      CALL FC    48 (
           UnitNo                   := #UnitNo,
           PrId                     := #Prid,
           Run                      := DB1941.DBX   17.4,
           PrIdTransfer             := TRUE,
           Start                    := TRUE,
           RetVal                   := #wRetVal);
Strt: NOP   0;

      L     0;
      T     DB502.DBD  156;

NETWORK
TITLE =external releases

      SET   ;
      =     DB2940.DBX  106.7;
      =     DB2940.DBX  266.7;
      =     DB2940.DBX  346.7;
      =     DB2940.DBX  426.7;
      =     DB2940.DBX  506.7;
      =     DB2940.DBX  586.7;
      =     DB2940.DBX  666.7;
      =     DB2940.DBX  746.7;
      =     DB2940.DBX  826.7;
      =     DB2940.DBX  906.7;
      =     DB2940.DBX  986.7;
      =     DB2940.DBX 1066.7;
      =     DB2940.DBX 1146.7;
      =     DB2940.DBX 1226.7;
      =     DB2940.DBX 1306.7;
      =     DB2940.DBX 1386.7;
      =     DB2940.DBX 1466.7;
      =     DB2940.DBX 1546.7;
NETWORK
TITLE =write own unit data

      SET   ;

//-- CIP Communication ---------------------------------------
      AN    DB1941.DBX   15.0;
      AN    DB1941.DBX 1233.6; // CIP Active (Slave)
      A     #ComCIP;
      JCN   NCIP;
//Conductivity CIP Return
      L     DB1945.DBD  150;
      T     DB1941.DBD  626;

//Temperature CIP Return
      L     DB1945.DBD  146;
      T     DB1941.DBD  594;

//CIP Prerun Pump SP
      CALL FC    45 (
           SFM                      := DB1941.DBD  686,
           Indexes                  := #SFM36);


      L     0.000000e+000;
      A     #SFM36.I01;
      =     DB1945.DBX  171.7;
      JCN   pfc;
      L     DB1941.DBD  654;
pfc:  NOP   0;
      A     #SFM36.I02;
      =     DB1945.DBX  172.0;
      JCN   ppc;
      L     DB1941.DBD  670;
ppc:  NOP   0;
      A     #SFM36.I03;
      =     DB1945.DBX  171.6;
      JCN   pxc;
      L     DB1941.DBD  574;
pxc:  NOP   0;
      T     DB1945.DBD  182;

//CIP Return
      L     DB1941.DBD  558;
      T     DB1945.DBD  186;
      L     DB1945.DBD  138;
      T     DB1941.DBD  562;

//CIP Prerun
      L     DB1941.DBD  542;
      T     DB1945.DBD  190;
      L     DB1945.DBD  142;
      T     DB1941.DBD  546;

// CIP Prerun Temperature
      L     DB1941.DBD  686;
      T     DB1945.DBD  182;

// Write Own Data to CIP
      L     DB1945.DBD   10;
      T     DB1945.DBD  154;

      L     DB1945.DBW   14;
      T     DB1945.DBW  158;

      L     DB1945.DBW   16;
      T     DB1945.DBW  160;

      L     DB1945.DBW   18;
      T     DB1945.DBW  162;

      L     DB1945.DBW   20;
      T     DB1945.DBW  164;

      L     DB1945.DBW   22;
      T     DB1945.DBW  166;

      A     DB1945.DBX   24.0;
      =     DB1945.DBX  168.0;

      A     DB1945.DBX   24.1;
      =     DB1945.DBX  168.1;

      A     DB1945.DBX   24.2;
      =     DB1945.DBX  168.2;

      A     DB1945.DBX   24.3;
      =     DB1945.DBX  168.3;

      A     DB1945.DBX   24.4;
      =     DB1945.DBX  168.4;

      A     DB1945.DBX   24.5;
      =     DB1945.DBX  168.5;

      A     DB1945.DBX   24.6;
      =     DB1945.DBX  168.6;

      A     DB1945.DBX   24.7;
      =     DB1945.DBX  168.7;

      L     DB1945.DBD  138; // CIP Amount
      T     DB1945.DBD   54; // CIP Amount

// Copy Data to CIP
      CALL SFC   20 (
           SRCBLK                   := DB1945.ToCIP,
           RET_VAL                  := #iRetVal,
           DSTBLK                   := DB502.ToCIP1);

      CLR   ;
      =     DB1945.DBX  173.7;

NCIP: NOP   0;

//Empty Signal
//A     "U094SpID".SpI.Sig //!!!! Insert correct Empty Signal !!!
      CLR   ;
      =     DB1945.DBX   26.5;

//Full Signal
//A     "U094SpID".SpI.Sig //!!!! Insert correct Full Signal !!!
      CLR   ;
      =     DB1945.DBX   26.2;

//CIP Program Selected
      A     #CIP;
      =     DB1945.DBX   27.1;

// Emergency Stop
      A     #EStopOK; //If needed add or replace with own SpI
      =     DB1945.DBX   27.0; //Emergency Stop OK


NETWORK
TITLE = read from other unit data



END_FUNCTION_BLOCK

FUNCTION_BLOCK FB 1949
TITLE =U094: CIP 1 Distribution
AUTHOR : Woermann
FAMILY : BOTEC_F1
NAME : Sim
VERSION : 0.1


VAR_TEMP
  CIP : BOOL ;	//CIP active
  xTmp : BOOL ;	//Temporary BOOL (free for general use)
  iTmp : INT ;	//Temporary INT (free for general use)
  rTmp : REAL ;	//Temporary REAL (free for general use)
  UnitNo : INT ;	//Unit Number
END_VAR
BEGIN
NETWORK
TITLE =General

      SET   ;
// get unit number ----------------------------------------------------------
      L     DB1940.DBW    0;
      T     #UnitNo;

// CIP ----------------------------------------------------------------------
      L     DB1941.DBD   54;
      L     0;
      <D    ;
      =     #CIP;

NETWORK
TITLE =Actuator

      A     DB1941.DBX   17.3;
      =     DB2940.DBX  105.3;
      =     DB2940.DBX  265.3;
      =     DB2940.DBX  345.3;
      =     DB2940.DBX  425.3;
      =     DB2940.DBX  505.3;
      =     DB2940.DBX  585.3;
      =     DB2940.DBX  665.3;
      =     DB2940.DBX  745.3;
      =     DB2940.DBX  825.3;
      =     DB2940.DBX  905.3;
      =     DB2940.DBX  985.3;
      =     DB2940.DBX 1065.3;
      =     DB2940.DBX 1145.3;
      =     DB2940.DBX 1225.3;
      =     DB2940.DBX 1305.3;
      =     DB2940.DBX 1385.3;
      =     DB2940.DBX 1465.3;
      =     DB2940.DBX 1545.3;


NETWORK
TITLE =Special Input

      A     DB1941.DBX   17.3;
      =     DB2941.DBX   81.3;
      =     DB2941.DBX  141.3;
      =     DB2941.DBX  201.3;
      =     DB2941.DBX  261.3;
      =     DB2941.DBX  321.3;
      =     DB2941.DBX  381.3;

NETWORK
TITLE =Counter

      A     DB1941.DBX   17.3;
      A     M    101.0;


      CLR   ;
NETWORK
TITLE =Analog Input

      A     DB1941.DBX   17.3;

NETWORK
TITLE =Universal Value

      A     DB1941.DBX   17.3;
//      =     "U094UnVD".unv001.Sim;
//      =     "U094UnVD".unv002.Sim;
//      =     "U094UnVD".RK1_KreisNr.Sim
//      =     "U094UnVD".RK1_Medium.Sim

NETWORK
TITLE =PID

      A     DB1941.DBX   17.3;

NETWORK
TITLE =Message

      A     DB1941.DBX   17.3;
//      =     "U094MsgD".msg001.Sim;
//      =     "U094MsgD".msg002.Sim;

NETWORK
TITLE =VLT

      A     DB1941.DBX   17.3;

END_FUNCTION_BLOCK

FUNCTION_BLOCK FB 1955
TITLE =U095: CIP 2 Distribution
FAMILY : BOTEC_F1
NAME : Comm
VERSION : 0.1


VAR_TEMP
  iRetVal : INT ;	//return value as integer
  wRetVal : WORD ;	//return value as word
  Run : BOOL ;	//Unit in "RUN" mode
  EStopOK : BOOL ;	//Emergency Stop OK
  CIP : BOOL ;	//CIP Program Selected
  ComCIP : BOOL ;	//Communication with CIP Active
  xTmp : BOOL ;	//Temporary BOOL (free for general use)
  iTmp : INT ;	//Temporary INT (free for general use)
  rTmp : REAL ;	//Temporary REAL (free for general use)
  dTmp : DINT ;	//Temporary DINT (free for general use)
  UnitNo : INT ;	//Unit Number
  EquipmentID : INT ;	//Equipment ID
  Prid : DINT ;	//Process ID
  SFM36 : STRUCT 	// CIP Pump Mode
   I00 : BOOL ;	// Off
   I01 : BOOL ;	// Flow
   I02 : BOOL ;	// Pressure
   I03 : BOOL ;	// Fix Speed
   I04 : BOOL ;
   I05 : BOOL ;
   I06 : BOOL ;
   I07 : BOOL ;
   I08 : BOOL ;
   I09 : BOOL ;
   I10 : BOOL ;
   I11 : BOOL ;
   I12 : BOOL ;
   I13 : BOOL ;
   I14 : BOOL ;
   I15 : BOOL ;
   I16 : BOOL ;
   I17 : BOOL ;
   I18 : BOOL ;
   I19 : BOOL ;
   I20 : BOOL ;
   I21 : BOOL ;
   I22 : BOOL ;
   I23 : BOOL ;
   I24 : BOOL ;
   I25 : BOOL ;
   I26 : BOOL ;
   I27 : BOOL ;
   I28 : BOOL ;
   I29 : BOOL ;
   I30 : BOOL ;
   I31 : BOOL ;
  END_STRUCT ;
END_VAR
BEGIN
NETWORK
TITLE =general

      SET   ;

// unit & equipment number ---------------------------------------------------
      L     DB1950.DBW    0;
      T     #UnitNo;

      L     DB1955.DBW   14;
      L     1000;
      *I    ;
      L     #UnitNo;
      +I    ;
      T     #EquipmentID;

// CIP ----------------------------------------------------------------------
      L     DB1955.DBW   18;
      L     0;
      <I    ;
      =     #CIP;

// Communicating Units-------------------------------------------------------
      L     DB1955.DBD   10;
      L     DB1955.DBD  106;
      ==D   ;
      =     #ComCIP;

// emergency OK -------------------------------------------------------------
      A     DB1955.DBX   75.0; //General Emergency Stop OK
      =     #EStopOK;

NETWORK
TITLE =read other unit's data

      SET   ;

// ... General Unit ----------/

      CALL FC   563 (
           ActReq                   := M    101.0,
           PLCNo                    := DB1955.DBW   14,
           SourceUnitNo             := 99,
           IsTUnit                  := FALSE,
           DstComDRec               := DB1955.GEN,
           RET_VAL                  := #wRetVal);


// ... CIP Unit ------------- /

      CALL FC   563 (
           ActReq                   := M    101.0,
           PLCNo                    := 3,
           SourceUnitNo             := 92,
           IsTUnit                  := FALSE,
           DstComDRec               := DB1955.CIP,
           RET_VAL                  := #wRetVal);

// ... To CIP Unit ------------- /
      AN    DB1951.DBX   15.0;
      A     DB1951.DBX 1233.6; // CIP Active (Slave)
      O     DB1951.DBX 1230.3; // production active
//    A     #ComCIP
      JCN   Slav;
      CALL SFC   20 (
           SRCBLK                   := DB502.ToCIP2,
           RET_VAL                  := #iRetVal,
           DSTBLK                   := DB1955.ToCIP);
Slav: NOP   0;

NETWORK
TITLE =remote start

      SET   ;

//-----------------------------------
// Start Request
//-----------------------------------
      L     DB502.DBD  160;
      L     0;
      >D    ;
      A     DB1951.DBX   15.0;
      A     DB1951.DBX   17.4;
      JCN   Strt;
      L     DB502.DBD  160;
      T     #Prid;

      CALL FC    48 (
           UnitNo                   := #UnitNo,
           PrId                     := #Prid,
           Run                      := DB1951.DBX   17.4,
           PrIdTransfer             := TRUE,
           Start                    := TRUE,
           RetVal                   := #wRetVal);
Strt: NOP   0;

      L     0;
      T     DB502.DBD  160;


NETWORK
TITLE =external releases

      SET   ;
      =     DB2950.DBX  266.7;
      =     DB2950.DBX  346.7;
      =     DB2950.DBX  506.7;
      =     DB2950.DBX  586.7;
NETWORK
TITLE =write own unit data

      SET   ;

//-- CIP Communication ---------------------------------------
      AN    DB1951.DBX   15.0;
      AN    DB1951.DBX 1233.6; // CIP Active (Slave)
      A     #ComCIP;
      JCN   NCIP;
//Conductivity CIP Return
      L     DB1955.DBD  150;
      T     DB1951.DBD  626;

//Temperature CIP Return
      L     DB1955.DBD  146;
      T     DB1951.DBD  594;

//CIP Prerun Pump SP
      CALL FC    45 (
           SFM                      := DB1951.DBD  686,
           Indexes                  := #SFM36);


      L     0.000000e+000;
      A     #SFM36.I01;
      =     DB1955.DBX  171.7;
      JCN   pfc;
      L     DB1951.DBD  654;
pfc:  NOP   0;
      A     #SFM36.I02;
      =     DB1955.DBX  172.0;
      JCN   ppc;
      L     DB1951.DBD  670;
ppc:  NOP   0;
      A     #SFM36.I03;
      =     DB1955.DBX  171.6;
      JCN   pxc;
      L     DB1951.DBD  574;
pxc:  NOP   0;
      T     DB1955.DBD  182;

//CIP Return
      L     DB1951.DBD  558;
      T     DB1955.DBD  186;
      L     DB1955.DBD  138;
      T     DB1951.DBD  562;

//CIP Prerun
      L     DB1951.DBD  542;
      T     DB1955.DBD  190;
      L     DB1955.DBD  142;
      T     DB1951.DBD  546;

// CIP Prerun Temperature
      L     DB1951.DBD  686;
      T     DB1955.DBD  182;

// Write Own Data to CIP
      L     DB1955.DBD   10;
      T     DB1955.DBD  154;

      L     DB1955.DBW   14;
      T     DB1955.DBW  158;

      L     DB1955.DBW   16;
      T     DB1955.DBW  160;

      L     DB1955.DBW   18;
      T     DB1955.DBW  162;

      L     DB1955.DBW   20;
      T     DB1955.DBW  164;

      L     DB1955.DBW   22;
      T     DB1955.DBW  166;

      A     DB1955.DBX   24.0;
      =     DB1955.DBX  168.0;

      A     DB1955.DBX   24.1;
      =     DB1955.DBX  168.1;

      A     DB1955.DBX   24.2;
      =     DB1955.DBX  168.2;

      A     DB1955.DBX   24.3;
      =     DB1955.DBX  168.3;

      A     DB1955.DBX   24.4;
      =     DB1955.DBX  168.4;

      A     DB1955.DBX   24.5;
      =     DB1955.DBX  168.5;

      A     DB1955.DBX   24.6;
      =     DB1955.DBX  168.6;

      A     DB1955.DBX   24.7;
      =     DB1955.DBX  168.7;

      L     DB1955.DBD  138; // CIP Amount
      T     DB1955.DBD   54; // CIP Amount

// Copy Data to CIP
      CALL SFC   20 (
           SRCBLK                   := DB1955.ToCIP,
           RET_VAL                  := #iRetVal,
           DSTBLK                   := DB502.ToCIP2);

NCIP: NOP   0;

//Empty Signal
//A     "U095SpID".SpI.Sig //!!!! Insert correct Empty Signal !!!
      CLR   ;
      =     DB1955.DBX   26.5;

//Full Signal
//A     "U095SpID".SpI.Sig //!!!! Insert correct Full Signal !!!
      CLR   ;
      =     DB1955.DBX   26.2;

//CIP Program Selected
      A     #CIP;
      =     DB1955.DBX   27.1;

// Emergency Stop
      A     #EStopOK; //If needed add or replace with own SpI
      =     DB1955.DBX   27.0; //Emergency Stop OK


NETWORK
TITLE = read from other unit data



END_FUNCTION_BLOCK

FUNCTION_BLOCK FB 1959
TITLE =U095: CIP 2 Distribution
AUTHOR : Woermann
FAMILY : BOTEC_F1
NAME : Sim
VERSION : 0.1


VAR_TEMP
  CIP : BOOL ;	//CIP active
  xTmp : BOOL ;	//Temporary BOOL (free for general use)
  iTmp : INT ;	//Temporary INT (free for general use)
  rTmp : REAL ;	//Temporary REAL (free for general use)
  UnitNo : INT ;	//Unit Number
END_VAR
BEGIN
NETWORK
TITLE =General

      SET   ;
// get unit number ----------------------------------------------------------
      L     DB1950.DBW    0;
      T     #UnitNo;

// CIP ----------------------------------------------------------------------
      L     DB1951.DBD   54;
      L     0;
      <D    ;
      =     #CIP;

NETWORK
TITLE =Actuator

      A     DB1951.DBX   17.3;
      =     DB2950.DBX  265.3;
      =     DB2950.DBX  345.3;
      =     DB2950.DBX  505.3;
      =     DB2950.DBX  585.3;
NETWORK
TITLE =Special Input

      A     DB1951.DBX   17.3;
      =     DB2951.DBX   81.3;
      =     DB2951.DBX  141.3;
      =     DB2951.DBX  201.3;
      =     DB2951.DBX  261.3;
NETWORK
TITLE =Counter

      A     DB1951.DBX   17.3;
      A     M    101.0;


      CLR   ;
NETWORK
TITLE =Analog Input

      A     DB1951.DBX   17.3;

NETWORK
TITLE =Universal Value

      A     DB1951.DBX   17.3;
//      =     "U095UnVD".unv001.Sim;
//      =     "U095UnVD".unv002.Sim;
//      =     "U095UnVD".RK2_KreisNr.Sim;
//      =     "U095UnVD".RK2_Medium.Sim;

NETWORK
TITLE =PID

      A     DB1951.DBX   17.3;

NETWORK
TITLE =Message

      A     DB1951.DBX   17.3;
//      =     "U095MsgD".msg001.Sim;
//      =     "U095MsgD".msg002.Sim;

NETWORK
TITLE =VLT

      A     DB1951.DBX   17.3;

END_FUNCTION_BLOCK

FUNCTION_BLOCK FB 1965
TITLE =U096: CIP 3 Distribution
FAMILY : BOTEC_F1
NAME : Comm
VERSION : 0.1


VAR_TEMP
  iRetVal : INT ;	//return value as integer
  wRetVal : WORD ;	//return value as word
  Run : BOOL ;	//Unit in "RUN" mode
  EStopOK : BOOL ;	//Emergency Stop OK
  CIP : BOOL ;	//CIP Program Selected
  ComCIP : BOOL ;	//Communication with CIP Active
  xTmp : BOOL ;	//Temporary BOOL (free for general use)
  iTmp : INT ;	//Temporary INT (free for general use)
  rTmp : REAL ;	//Temporary REAL (free for general use)
  dTmp : DINT ;	//Temporary DINT (free for general use)
  UnitNo : INT ;	//Unit Number
  EquipmentID : INT ;	//Equipment ID
  Prid : DINT ;	//Process ID
  SFM36 : STRUCT 	// CIP Pump Mode
   I00 : BOOL ;	// Off
   I01 : BOOL ;	// Flow
   I02 : BOOL ;	// Pressure
   I03 : BOOL ;	// Fix Speed
   I04 : BOOL ;
   I05 : BOOL ;
   I06 : BOOL ;
   I07 : BOOL ;
   I08 : BOOL ;
   I09 : BOOL ;
   I10 : BOOL ;
   I11 : BOOL ;
   I12 : BOOL ;
   I13 : BOOL ;
   I14 : BOOL ;
   I15 : BOOL ;
   I16 : BOOL ;
   I17 : BOOL ;
   I18 : BOOL ;
   I19 : BOOL ;
   I20 : BOOL ;
   I21 : BOOL ;
   I22 : BOOL ;
   I23 : BOOL ;
   I24 : BOOL ;
   I25 : BOOL ;
   I26 : BOOL ;
   I27 : BOOL ;
   I28 : BOOL ;
   I29 : BOOL ;
   I30 : BOOL ;
   I31 : BOOL ;
  END_STRUCT ;
END_VAR
BEGIN
NETWORK
TITLE =general

      SET   ;

// unit & equipment number ---------------------------------------------------
      L     DB1960.DBW    0;
      T     #UnitNo;

      L     DB1965.DBW   14;
      L     1000;
      *I    ;
      L     #UnitNo;
      +I    ;
      T     #EquipmentID;

// CIP ----------------------------------------------------------------------
      L     DB1965.DBW   18;
      L     0;
      <I    ;
      =     #CIP;

// Communicating Units-------------------------------------------------------
      L     DB1965.DBD   10;
      L     DB1965.DBD  106;
      ==D   ;
      =     #ComCIP;

// emergency OK -------------------------------------------------------------
      A     DB1965.DBX   75.0; //General Emergency Stop OK
      =     #EStopOK;

NETWORK
TITLE =read other unit's data

      SET   ;

// ... General Unit ----------/

      CALL FC   563 (
           ActReq                   := M    101.0,
           PLCNo                    := DB1965.DBW   14,
           SourceUnitNo             := 99,
           IsTUnit                  := FALSE,
           DstComDRec               := DB1965.GEN,
           RET_VAL                  := #wRetVal);


// ... CIP Unit ------------- /

      CALL FC   563 (
           ActReq                   := M    101.0,
           PLCNo                    := 3,
           SourceUnitNo             := 93,
           IsTUnit                  := FALSE,
           DstComDRec               := DB1965.CIP,
           RET_VAL                  := #wRetVal);

// ... To CIP Unit ------------- /
      A     DB1961.DBX 1233.6; // CIP Active (Slave)
      O     DB1961.DBX 1230.3; // production active
      AN    DB1961.DBX   15.0;

// A     #ComCIP
      JCN   Slav;
      CALL SFC   20 (
           SRCBLK                   := DB502.ToCIP3,
           RET_VAL                  := #iRetVal,
           DSTBLK                   := DB1965.ToCIP);
Slav: NOP   0;
NETWORK
TITLE =remote start

      SET   ;

//-----------------------------------
// Start Request
//-----------------------------------
      L     DB502.DBD  164;
      L     0;
      >D    ;
      A     DB1961.DBX   15.0;
      A     DB1961.DBX   17.4;
      JCN   Strt;
      L     DB502.DBD  164;
      T     #Prid;

      CALL FC    48 (
           UnitNo                   := #UnitNo,
           PrId                     := #Prid,
           Run                      := DB1961.DBX   17.4,
           PrIdTransfer             := TRUE,
           Start                    := TRUE,
           RetVal                   := #wRetVal);
Strt: NOP   0;

      L     0;
      T     DB502.DBD  164;


NETWORK
TITLE =external releases

      SET   ;
      =     DB2960.DBX  186.7;
      =     DB2960.DBX  266.7;
      =     DB2960.DBX  346.7;
      =     DB2960.DBX  426.7;
      =     DB2960.DBX  506.7;
      =     DB2960.DBX  586.7;
      =     DB2960.DBX  666.7;
      =     DB2960.DBX  746.7;
      =     DB2960.DBX  826.7;
      =     DB2960.DBX  906.7;
      =     DB2960.DBX  986.7;
      =     DB2960.DBX 1066.7;
      =     DB2960.DBX 1146.7;
      =     DB2960.DBX 1226.7;
      =     DB2960.DBX 1306.7;
      =     DB2960.DBX 1546.7;
NETWORK
TITLE =write own unit data

      SET   ;

//-- CIP Communication ---------------------------------------
      AN    DB1961.DBX   15.0;
      AN    DB1961.DBX 1233.6; // CIP Active (Slave)
      A     #ComCIP;
      JCN   NCIP;
//Conductivity CIP Return
      L     DB1965.DBD  150;
      T     DB1961.DBD  626;

//Temperature CIP Return
      L     DB1965.DBD  146;
      T     DB1961.DBD  594;

//CIP Prerun Pump SP

      CALL FC    45 (
           SFM                      := DB1961.DBD  686,
           Indexes                  := #SFM36);


      L     0.000000e+000;
      A     #SFM36.I01;
      =     DB1965.DBX  171.7;
      JCN   pfc;
      L     DB1961.DBD  654;
pfc:  NOP   0;
      A     #SFM36.I02;
      =     DB1965.DBX  172.0;
      JCN   ppc;
      L     DB1961.DBD  670;
ppc:  NOP   0;
      A     #SFM36.I03;
      =     DB1965.DBX  171.6;
      JCN   pxc;
      L     DB1961.DBD  574;
pxc:  NOP   0;
      T     DB1965.DBD  182;

//CIP Return
      L     DB1961.DBD  558;
      T     DB1965.DBD  186;
      L     DB1965.DBD  138;
      T     DB1961.DBD  562;

//CIP Prerun
      L     DB1961.DBD  542;
      T     DB1965.DBD  190;
      L     DB1965.DBD  142;
      T     DB1961.DBD  546;

// CIP Prerun Temperature
      L     DB1961.DBD  686;
      T     DB1965.DBD  182;

// Write Own Data to CIP
      L     DB1965.DBD   10;
      T     DB1965.DBD  154;

      L     DB1965.DBW   14;
      T     DB1965.DBW  158;

      L     DB1965.DBW   16;
      T     DB1965.DBW  160;

      L     DB1965.DBW   18;
      T     DB1965.DBW  162;

      L     DB1965.DBW   20;
      T     DB1965.DBW  164;

      L     DB1965.DBW   22;
      T     DB1965.DBW  166;

      A     DB1965.DBX   24.0;
      =     DB1965.DBX  168.0;

      A     DB1965.DBX   24.1;
      =     DB1965.DBX  168.1;

      A     DB1965.DBX   24.2;
      =     DB1965.DBX  168.2;

      A     DB1965.DBX   24.3;
      =     DB1965.DBX  168.3;

      A     DB1965.DBX   24.4;
      =     DB1965.DBX  168.4;

      A     DB1965.DBX   24.5;
      =     DB1965.DBX  168.5;

      A     DB1965.DBX   24.6;
      =     DB1965.DBX  168.6;

      A     DB1965.DBX   24.7;
      =     DB1965.DBX  168.7;

      L     DB1965.DBD  138; // CIP Amount
      T     DB1965.DBD   54; // CIP Amount

// Copy Data to CIP
      CALL SFC   20 (
           SRCBLK                   := DB1965.ToCIP,
           RET_VAL                  := #iRetVal,
           DSTBLK                   := DB502.ToCIP3);

NCIP: NOP   0;

//Empty Signal
//A     "U096SpID".SpI.Sig //!!!! Insert correct Empty Signal !!!
      CLR   ;
      =     DB1965.DBX   26.5;

//Full Signal
//A     "U096SpID".SpI.Sig //!!!! Insert correct Full Signal !!!
      CLR   ;
      =     DB1965.DBX   26.2;

//CIP Program Selected
      A     #CIP;
      =     DB1965.DBX   27.1;

// Emergency Stop
      A     #EStopOK; //If needed add or replace with own SpI
      =     DB1965.DBX   27.0; //Emergency Stop OK


NETWORK
TITLE = read from other unit data



END_FUNCTION_BLOCK

FUNCTION_BLOCK FB 1969
TITLE =U096: CIP 3 Distribution
AUTHOR : Woermann
FAMILY : BOTEC_F1
NAME : Sim
VERSION : 0.1


VAR_TEMP
  CIP : BOOL ;	//CIP active
  xTmp : BOOL ;	//Temporary BOOL (free for general use)
  iTmp : INT ;	//Temporary INT (free for general use)
  rTmp : REAL ;	//Temporary REAL (free for general use)
  UnitNo : INT ;	//Unit Number
END_VAR
BEGIN
NETWORK
TITLE =General

      SET   ;
// get unit number ----------------------------------------------------------
      L     DB1960.DBW    0;
      T     #UnitNo;

// CIP ----------------------------------------------------------------------
      L     DB1961.DBD   54;
      L     0;
      <D    ;
      =     #CIP;

NETWORK
TITLE =Actuator

      A     DB1961.DBX   17.3;
      =     DB2960.DBX  185.3;
      =     DB2960.DBX  265.3;
      =     DB2960.DBX  345.3;
      =     DB2960.DBX  425.3;
      =     DB2960.DBX  505.3;
      =     DB2960.DBX  585.3;
      =     DB2960.DBX  665.3;
      =     DB2960.DBX  745.3;
      =     DB2960.DBX  825.3;
      =     DB2960.DBX  905.3;
      =     DB2960.DBX  985.3;
      =     DB2960.DBX 1065.3;
      =     DB2960.DBX 1145.3;
      =     DB2960.DBX 1225.3;
      =     DB2960.DBX 1305.3;
      =     DB2960.DBX 1545.3;
NETWORK
TITLE =Special Input

      A     DB1961.DBX   17.3;
      =     DB2961.DBX   81.3;
      =     DB2961.DBX  141.3;
      =     DB2961.DBX  201.3;
      =     DB2961.DBX  261.3;
      =     DB2961.DBX  321.3;
      =     DB2961.DBX  381.3;

NETWORK
TITLE =Counter

      A     DB1961.DBX   17.3;
      A     M    101.0;
      CLR   ;
NETWORK
TITLE =Analog Input

      A     DB1961.DBX   17.3;

NETWORK
TITLE =Universal Value

      A     DB1961.DBX   17.3;
//      =     "U096UnVD".unv001.Sim;
//      =     "U096UnVD".unv002.Sim;
//      =     "U096UnVD".RK3_KreisNr.Sim;
//      =     "U096UnVD".RK3_Medium.Sim;

NETWORK
TITLE =PID

      A     DB1961.DBX   17.3;

NETWORK
TITLE =Message

      A     DB1961.DBX   17.3;
//      =     "U096MsgD".msg001.Sim;
//      =     "U096MsgD".msg002.Sim;

NETWORK
TITLE =VLT

      A     DB1961.DBX   17.3;

END_FUNCTION_BLOCK

FUNCTION_BLOCK FB 1985
TITLE =U098: General Syrup Room
FAMILY : BOTEC_F1
NAME : Comm
VERSION : 0.1


VAR_TEMP
  iRetVal : INT ;	//return value as integer
  wRetVal : WORD ;	//return value as word
  Run : BOOL ;	//Unit in "RUN" mode
  EStopOK : BOOL ;	//Emergency Stop OK
  CIP : BOOL ;	//CIP Program Selected
  ComCIP : BOOL ;	//Communication with CIP Active
  xTmp : BOOL ;	//Temporary BOOL (free for general use)
  iTmp : INT ;	//Temporary INT (free for general use)
  rTmp : REAL ;	//Temporary REAL (free for general use)
  dTmp : DINT ;	//Temporary DINT (free for general use)
  UnitNo : INT ;	//Unit Number
  EquipmentID : INT ;	//Equipment ID
  Prid : DINT ;	//Process ID
  SFM36 : STRUCT 	// CIP Pump Mode
   I00 : BOOL ;	// Off
   I01 : BOOL ;	// Flow
   I02 : BOOL ;	// Pressure
   I03 : BOOL ;	// Fix Speed
   I04 : BOOL ;
   I05 : BOOL ;
   I06 : BOOL ;
   I07 : BOOL ;
   I08 : BOOL ;
   I09 : BOOL ;
   I10 : BOOL ;
   I11 : BOOL ;
   I12 : BOOL ;
   I13 : BOOL ;
   I14 : BOOL ;
   I15 : BOOL ;
   I16 : BOOL ;
   I17 : BOOL ;
   I18 : BOOL ;
   I19 : BOOL ;
   I20 : BOOL ;
   I21 : BOOL ;
   I22 : BOOL ;
   I23 : BOOL ;
   I24 : BOOL ;
   I25 : BOOL ;
   I26 : BOOL ;
   I27 : BOOL ;
   I28 : BOOL ;
   I29 : BOOL ;
   I30 : BOOL ;
   I31 : BOOL ;
  END_STRUCT ;
END_VAR
BEGIN
NETWORK
TITLE =general

      SET   ;

// unit & equipment number ---------------------------------------------------
      L     DB1980.DBW    0;
      T     #UnitNo;

      L     DB1985.DBW   14;
      L     1000;
      *I    ;
      L     #UnitNo;
      +I    ;
      T     #EquipmentID;

// CIP ----------------------------------------------------------------------
      L     DB1985.DBW   18;
      L     0;
      <I    ;
      =     #CIP;

// Communicating Units-------------------------------------------------------
      L     DB1985.DBD   10;
      L     DB1985.DBD  106;
      ==D   ;
      =     #ComCIP;

// emergency OK -------------------------------------------------------------
      A     DB1985.DBX   75.0; //General Emergency Stop OK
      =     #EStopOK;

NETWORK
TITLE =read other unit's data

      SET   ;

// ... General Unit ----------/

      CALL FC   563 (
           ActReq                   := M    101.0,
           PLCNo                    := DB1985.DBW   14,
           SourceUnitNo             := 99,
           IsTUnit                  := FALSE,
           DstComDRec               := DB1985.GEN,
           RET_VAL                  := #wRetVal);


NETWORK
TITLE =remote start

      SET   ;
// !!! insert correct condition of unit start !!!
      A     DB1981.DBX   15.0;
      A     DB1981.DBX   17.4;
      CLR   ;
      JCN   Strt;
      L     DB1985.DBD   10;
//L        L#-1;                            // Prid negative to start on its own
      T     #Prid;

      CALL FC    48 (
           UnitNo                   := #UnitNo,
           PrId                     := #Prid,
           Run                      := DB1981.DBX   17.4,
           PrIdTransfer             := TRUE,
           Start                    := TRUE,
           RetVal                   := #wRetVal);
Strt: NOP   0;
NETWORK
TITLE =external releases

      SET   ;
      =     DB2980.DBX  106.7;
      =     DB2980.DBX  186.7;
      =     DB2980.DBX  266.7;
      =     DB2980.DBX  346.7;
      =     DB2980.DBX  426.7;
      =     DB2980.DBX  506.7;
      =     DB2980.DBX  586.7;
      =     DB2980.DBX  666.7;
NETWORK
TITLE =write own unit data

      SET   ;

//-- CIP Communication ---------------------------------------
      AN    DB1981.DBX   15.0;
//      AN "U098SeqD".Seq.PO.B30 // CIP Active (Slave)
      A     #ComCIP;
      JCN   NCIP;
//Conductivity CIP Return
      L     DB1985.DBD  150;
      T     DB1981.DBD  626;

//Temperature CIP Return
      L     DB1985.DBD  146;
      T     DB1981.DBD  594;

//CIP Prerun Pump SP

      CALL FC    45 (
           SFM                      := DB1981.DBD  686,
           Indexes                  := #SFM36);


      L     0.000000e+000;
      A     #SFM36.I01;
      =     DB1985.DBX  171.7;
      JCN   pfc;
      L     DB1981.DBD  654;
pfc:  NOP   0;
      A     #SFM36.I02;
      =     DB1985.DBX  172.0;
      JCN   ppc;
      L     DB1981.DBD  670;
ppc:  NOP   0;
      A     #SFM36.I03;
      =     DB1985.DBX  171.6;
      JCN   pxc;
      L     DB1981.DBD  574;
pxc:  NOP   0;
      T     DB1985.DBD  182;

//CIP Return
      L     DB1981.DBD  558;
      T     DB1985.DBD  186;
      L     DB1985.DBD  138;
      T     DB1981.DBD  562;

//CIP Prerun
      L     DB1981.DBD  542;
      T     DB1985.DBD  190;
      L     DB1985.DBD  142;
      T     DB1981.DBD  546;

// Write Own Data to CIP
      L     DB1985.DBD   10;
      T     DB1985.DBD  154;

      L     DB1985.DBW   14;
      T     DB1985.DBW  158;

      L     DB1985.DBW   16;
      T     DB1985.DBW  160;

      L     DB1985.DBW   18;
      T     DB1985.DBW  162;

      L     DB1985.DBW   20;
      T     DB1985.DBW  164;

      L     DB1985.DBW   22;
      T     DB1985.DBW  166;

      A     DB1985.DBX   24.0;
      =     DB1985.DBX  168.0;

      A     DB1985.DBX   24.1;
      =     DB1985.DBX  168.1;

      A     DB1985.DBX   24.2;
      =     DB1985.DBX  168.2;

      A     DB1985.DBX   24.3;
      =     DB1985.DBX  168.3;

      A     DB1985.DBX   24.4;
      =     DB1985.DBX  168.4;

      A     DB1985.DBX   24.5;
      =     DB1985.DBX  168.5;

      A     DB1985.DBX   24.6;
      =     DB1985.DBX  168.6;

      A     DB1985.DBX   24.7;
      =     DB1985.DBX  168.7;

// Copy Data to CIP
      CALL SFC   20 (
           SRCBLK                   := DB1985.ToCIP,
           RET_VAL                  := #iRetVal,
           DSTBLK                   := DB1985.ToCIP);

NCIP: NOP   0;

//Empty Signal
//A     "U098SpID".SpI.Sig //!!!! Insert correct Empty Signal !!!
      CLR   ;
      =     DB1985.DBX   26.5;

//Full Signal
//A     "U098SpID".SpI.Sig //!!!! Insert correct Full Signal !!!
      CLR   ;
      =     DB1985.DBX   26.2;

//CIP Program Selected
      A     #CIP;
      =     DB1985.DBX   27.1;

// Emergency Stop
      A     #EStopOK; //If needed add or replace with own SpI
      =     DB1985.DBX   27.0; //Emergency Stop OK


NETWORK
TITLE = read from other unit data



END_FUNCTION_BLOCK

FUNCTION_BLOCK FB 1989
TITLE =U098: General Syrup Room
AUTHOR : Woermann
FAMILY : BOTEC_F1
NAME : Sim
VERSION : 0.1


VAR_TEMP
  CIP : BOOL ;	//CIP active
  xTmp : BOOL ;	//Temporary BOOL (free for general use)
  iTmp : INT ;	//Temporary INT (free for general use)
  rTmp : REAL ;	//Temporary REAL (free for general use)
  UnitNo : INT ;	//Unit Number
END_VAR
BEGIN
NETWORK
TITLE =General

      SET   ;
// get unit number ----------------------------------------------------------
      L     DB1980.DBW    0;
      T     #UnitNo;

// CIP ----------------------------------------------------------------------
      L     DB1981.DBD   54;
      L     0;
      <D    ;
      =     #CIP;

NETWORK
TITLE =Actuator

      A     DB1981.DBX   17.3;
      =     DB2980.DBX  105.3;
      =     DB2980.DBX  185.3;
      =     DB2980.DBX  265.3;
      =     DB2980.DBX  345.3;
      =     DB2980.DBX  425.3;
      =     DB2980.DBX  505.3;
      =     DB2980.DBX  585.3;
      =     DB2980.DBX  665.3;

NETWORK
TITLE =Special Input

      A     DB1981.DBX   17.3;
      =     DB2981.DBX   81.3;
      =     DB2981.DBX  141.3;
      =     DB2981.DBX  201.3;
      =     DB2981.DBX  261.3;
      =     DB2981.DBX  321.3;
      =     DB2981.DBX  381.3;
      =     DB2981.DBX  441.3;
      =     DB2981.DBX  501.3;

NETWORK
TITLE =Counter

      A     DB1981.DBX   17.3;
      A     M    101.0;


      CLR   ;
NETWORK
TITLE =Analog Input

      A     DB1981.DBX   17.3;
      =     DB2983.DBX  141.3;
      =     DB2983.DBX  261.3;
      =     DB2983.DBX  381.3;
      =     DB2983.DBX  501.3;

NETWORK
TITLE =Universal Value

      A     DB1981.DBX   17.3;
//      =     "U098UnVD".unv001.Sim;
//      =     "U098UnVD".unv002.Sim;

NETWORK
TITLE =PID

      A     DB1981.DBX   17.3;

NETWORK
TITLE =Message

      A     DB1981.DBX   17.3;
//      =     "U098MsgD".msg001.Sim;
//      =     "U098MsgD".msg002.Sim;

NETWORK
TITLE =VLT

      A     DB1981.DBX   17.3;

END_FUNCTION_BLOCK

FUNCTION_BLOCK FB 1995
TITLE =U099: PLC 3 General
FAMILY : BOTEC_F1
NAME : Comm
VERSION : 0.1


VAR_TEMP
  iRetVal : INT ;	//return value as integer
  wRetVal : WORD ;	//return value as word
  Run : BOOL ;	//Unit in "RUN" mode
  EStopOK : BOOL ;	//Emergency Stop OK
  CIP : BOOL ;	//CIP Program Selected
  ComCIP : BOOL ;	//Communication with CIP Active
  xTmp : BOOL ;	//Temporary BOOL (free for general use)
  iTmp : INT ;	//Temporary INT (free for general use)
  rTmp : REAL ;	//Temporary REAL (free for general use)
  dTmp : DINT ;	//Temporary DINT (free for general use)
  UnitNo : INT ;	//Unit Number
  EquipmentID : INT ;	//Equipment ID
  Prid : DINT ;	//Process ID
  SFM36 : STRUCT 	// CIP Pump Mode
   I00 : BOOL ;	// Off
   I01 : BOOL ;	// Flow
   I02 : BOOL ;	// Pressure
   I03 : BOOL ;	// Fix Speed
   I04 : BOOL ;
   I05 : BOOL ;
   I06 : BOOL ;
   I07 : BOOL ;
   I08 : BOOL ;
   I09 : BOOL ;
   I10 : BOOL ;
   I11 : BOOL ;
   I12 : BOOL ;
   I13 : BOOL ;
   I14 : BOOL ;
   I15 : BOOL ;
   I16 : BOOL ;
   I17 : BOOL ;
   I18 : BOOL ;
   I19 : BOOL ;
   I20 : BOOL ;
   I21 : BOOL ;
   I22 : BOOL ;
   I23 : BOOL ;
   I24 : BOOL ;
   I25 : BOOL ;
   I26 : BOOL ;
   I27 : BOOL ;
   I28 : BOOL ;
   I29 : BOOL ;
   I30 : BOOL ;
   I31 : BOOL ;
  END_STRUCT ;
  SEND_DONE : BOOL ;
  SEND_ERROR : BOOL ;
  SEND_STATUS : WORD ;
  RECV_NDR : BOOL ;
  RECV_ERROR : BOOL ;
  RECV_STATUS : WORD ;
END_VAR
BEGIN
NETWORK
TITLE =general

      SET   ;

// unit & equipment number ---------------------------------------------------
      L     DB1990.DBW    0;
      T     #UnitNo;

      L     DB1995.DBW   14;
      L     1000;
      *I    ;
      L     #UnitNo;
      +I    ;
      T     #EquipmentID;

// CIP ----------------------------------------------------------------------
      L     DB1995.DBW   18;
      L     0;
      <I    ;
      =     #CIP;

// Communicating Units-------------------------------------------------------
      L     DB1995.DBD   10;
      L     DB1995.DBD  106;
      ==D   ;
      =     #ComCIP;

// emergency OK -------------------------------------------------------------
      A     DB1995.DBX   75.0; //General Emergency Stop OK
      =     #EStopOK;

NETWORK
TITLE =read other unit's data

      SET   ;

      L     MW  2900;
      SLW   1;
      T     MW  2900;
      L     0;
      ==D   ;
      S     M   2901.0;


// ... General Unit ----------/

      CALL FC   563 (
           ActReq                   := TRUE,
           PLCNo                    := DB1995.DBW   14,
           SourceUnitNo             := 99,
           IsTUnit                  := FALSE,
           DstComDRec               := DB1995.GEN,
           RET_VAL                  := #wRetVal);

// ... MTE1 from PLC01 ------------- /

      CALL FC   563 (
           ActReq                   := M    101.0,
           PLCNo                    := 1,
           SourceUnitNo             := 14,
           IsTUnit                  := FALSE,
           DstComDRec               := DB1995.MTE1,
           RET_VAL                  := #wRetVal);

// ... MTE2 from PLC01 ------------- /

      CALL FC   563 (
           ActReq                   := M    101.0,
           PLCNo                    := 1,
           SourceUnitNo             := 19,
           IsTUnit                  := FALSE,
           DstComDRec               := DB1995.MTE2,
           RET_VAL                  := #wRetVal);

// ... MTE3 from PLC01 ------------- /

      CALL FC   563 (
           ActReq                   := M    101.0,
           PLCNo                    := 1,
           SourceUnitNo             := 24,
           IsTUnit                  := FALSE,
           DstComDRec               := DB1995.MTE3,
           RET_VAL                  := #wRetVal);

// ... MTE4 from PLC01 ------------- /

      CALL FC   563 (
           ActReq                   := M    101.0,
           PLCNo                    := 1,
           SourceUnitNo             := 29,
           IsTUnit                  := FALSE,
           DstComDRec               := DB1995.MTE4,
           RET_VAL                  := #wRetVal);

// ... KZESR from PLC01 ------------- /

      CALL FC   563 (
           ActReq                   := M    101.0,
           PLCNo                    := 1,
           SourceUnitNo             := 7,
           IsTUnit                  := FALSE,
           DstComDRec               := DB1995.P01U007,
           RET_VAL                  := #wRetVal);

// ... Wasser SR from PLC01 ------------- /

      CALL FC   563 (
           ActReq                   := M    101.0,
           PLCNo                    := 1,
           SourceUnitNo             := 9,
           IsTUnit                  := FALSE,
           DstComDRec               := DB1995.P01U009,
           RET_VAL                  := #wRetVal);



//----------------------------------------
// Communication Remote Wells
//----------------------------------------

// ...Well Transfer A from PLC04 --- /
      CALL FC   563 (
           ActReq                   := M    101.0,
           PLCNo                    := 4,
           SourceUnitNo             := 25,
           IsTUnit                  := FALSE,
           DstComDRec               := DB1995.P04U025,
           RET_VAL                  := #wRetVal);

// ...Well Transfer B from PLC04 --- /
      CALL FC   563 (
           ActReq                   := M    101.0,
           PLCNo                    := 4,
           SourceUnitNo             := 26,
           IsTUnit                  := FALSE,
           DstComDRec               := DB1995.P04U026,
           RET_VAL                  := #wRetVal);

// ...Well Transfer CF from PLC04 --- /
      CALL FC   563 (
           ActReq                   := M    101.0,
           PLCNo                    := 4,
           SourceUnitNo             := 27,
           IsTUnit                  := FALSE,
           DstComDRec               := DB1995.P04U027,
           RET_VAL                  := #wRetVal);

// ...Well Transfer C from PLC04 --- /
      CALL FC   563 (
           ActReq                   := M    101.0,
           PLCNo                    := 4,
           SourceUnitNo             := 28,
           IsTUnit                  := FALSE,
           DstComDRec               := DB1995.P04U028,
           RET_VAL                  := #wRetVal);

// ...Well Transfer B6F from PLC04 --- /
      CALL FC   563 (
           ActReq                   := M    101.0,
           PLCNo                    := 4,
           SourceUnitNo             := 29,
           IsTUnit                  := FALSE,
           DstComDRec               := DB1995.P04U029,
           RET_VAL                  := #wRetVal);

// ...Well Transfer H6 from PLC04 --- /
      CALL FC   563 (
           ActReq                   := M    101.0,
           PLCNo                    := 4,
           SourceUnitNo             := 30,
           IsTUnit                  := FALSE,
           DstComDRec               := DB1995.P04U030,
           RET_VAL                  := #wRetVal);

// ...Well Transfer J6 from PLC04 --- /
      CALL FC   563 (
           ActReq                   := M    101.0,
           PLCNo                    := 4,
           SourceUnitNo             := 31,
           IsTUnit                  := FALSE,
           DstComDRec               := DB1995.P04U031,
           RET_VAL                  := #wRetVal);

// ...Well Transfer L6F from PLC04 --- /
      CALL FC   563 (
           ActReq                   := M    101.0,
           PLCNo                    := 4,
           SourceUnitNo             := 32,
           IsTUnit                  := FALSE,
           DstComDRec               := DB1995.P04U032,
           RET_VAL                  := #wRetVal);

// ...Well Transfer B6 from PLC04 --- /
      CALL FC   563 (
           ActReq                   := M    101.0,
           PLCNo                    := 4,
           SourceUnitNo             := 33,
           IsTUnit                  := FALSE,
           DstComDRec               := DB1995.P04U033,
           RET_VAL                  := #wRetVal);

// ...Well Transfer D6 from PLC04 --- /
      CALL FC   563 (
           ActReq                   := M    101.0,
           PLCNo                    := 4,
           SourceUnitNo             := 34,
           IsTUnit                  := FALSE,
           DstComDRec               := DB1995.P04U034,
           RET_VAL                  := #wRetVal);

//----------------------------------------
// Communication Local Wells
//----------------------------------------
// ...Local Well 2A from PLC04 --- /
      CALL FC   563 (
           ActReq                   := M    101.0,
           PLCNo                    := 4,
           SourceUnitNo             := 1,
           IsTUnit                  := FALSE,
           DstComDRec               := DB1995.P04U001,
           RET_VAL                  := #wRetVal);

// ...Local Well 2B from PLC04 --- /
      CALL FC   563 (
           ActReq                   := M    101.0,
           PLCNo                    := 4,
           SourceUnitNo             := 2,
           IsTUnit                  := FALSE,
           DstComDRec               := DB1995.P04U002,
           RET_VAL                  := #wRetVal);


// ...Local Well 3 from PLC04 --- /
      CALL FC   563 (
           ActReq                   := M    101.0,
           PLCNo                    := 4,
           SourceUnitNo             := 3,
           IsTUnit                  := FALSE,
           DstComDRec               := DB1995.P04U003,
           RET_VAL                  := #wRetVal);

// ...Local Well 7 from PLC04 --- /
      CALL FC   563 (
           ActReq                   := M    101.0,
           PLCNo                    := 4,
           SourceUnitNo             := 4,
           IsTUnit                  := FALSE,
           DstComDRec               := DB1995.P04U004,
           RET_VAL                  := #wRetVal);


//----------------------------------------
// Communication P01 Anlage
//----------------------------------------
      CALL FC   563 (
           ActReq                   := M    101.0,
           PLCNo                    := 1,
           SourceUnitNo             := 153,
           IsTUnit                  := FALSE,
           DstComDRec               := DB1995.P01U153,
           RET_VAL                  := #wRetVal);

      CALL FC   563 (
           ActReq                   := M    101.0,
           PLCNo                    := 1,
           SourceUnitNo             := 155,
           IsTUnit                  := FALSE,
           DstComDRec               := DB1995.P01U155,
           RET_VAL                  := #wRetVal);

      CALL FC   563 (
           ActReq                   := M    101.0,
           PLCNo                    := 1,
           SourceUnitNo             := 157,
           IsTUnit                  := FALSE,
           DstComDRec               := DB1995.P01U157,
           RET_VAL                  := #wRetVal);

      CALL FC   563 (
           ActReq                   := M    101.0,
           PLCNo                    := 1,
           SourceUnitNo             := 159,
           IsTUnit                  := FALSE,
           DstComDRec               := DB1995.P01U159,
           RET_VAL                  := #wRetVal);

      CALL FC   563 (
           ActReq                   := M    101.0,
           PLCNo                    := 1,
           SourceUnitNo             := 162,
           IsTUnit                  := FALSE,
           DstComDRec               := DB1995.P01U162,
           RET_VAL                  := #wRetVal);

      CALL FC   563 (
           ActReq                   := M    101.0,
           PLCNo                    := 1,
           SourceUnitNo             := 164,
           IsTUnit                  := FALSE,
           DstComDRec               := DB1995.P01U164,
           RET_VAL                  := #wRetVal);


NETWORK
TITLE =remote start

      SET   ;
// !!! insert correct condition of unit start !!!
      A     DB1991.DBX   15.0;
      A     DB1991.DBX   17.4;
      CLR   ;
      JCN   Strt;
      L     DB1995.DBD   10;
//L        L#-1;                            // Prid negative to start on its own
      T     #Prid;

      CALL FC    48 (
           UnitNo                   := #UnitNo,
           PrId                     := #Prid,
           Run                      := DB1991.DBX   17.4,
           PrIdTransfer             := TRUE,
           Start                    := TRUE,
           RetVal                   := #wRetVal);
Strt: NOP   0;
NETWORK
TITLE =external releases

      SET   ;
      =     DB2990.DBX  106.7;
      =     DB2990.DBX  186.7;
      =     DB2990.DBX  266.7;
NETWORK
TITLE =write own unit data

      SET   ;

//-- CIP Communication ---------------------------------------
      AN    DB1991.DBX   15.0;
//      AN "U099SeqD".Seq.PO.B30 // CIP Active (Slave)
      A     #ComCIP;
      JCN   NCIP;
//Conductivity CIP Return
      L     DB1995.DBD  150;
      T     DB1991.DBD  626;

//Temperature CIP Return
      L     DB1995.DBD  146;
      T     DB1991.DBD  594;

//CIP Prerun Pump SP

      CALL FC    45 (
           SFM                      := DB1991.DBD  686,
           Indexes                  := #SFM36);


      L     0.000000e+000;
      A     #SFM36.I01;
      =     DB1995.DBX  171.7;
      JCN   pfc;
      L     DB1991.DBD  654;
pfc:  NOP   0;
      A     #SFM36.I02;
      =     DB1995.DBX  172.0;
      JCN   ppc;
      L     DB1991.DBD  670;
ppc:  NOP   0;
      A     #SFM36.I03;
      =     DB1995.DBX  171.6;
      JCN   pxc;
      L     DB1991.DBD  574;
pxc:  NOP   0;
      T     DB1995.DBD  182;

//CIP Return
      L     DB1991.DBD  558;
      T     DB1995.DBD  186;
      L     DB1995.DBD  138;
      T     DB1991.DBD  562;

//CIP Prerun
      L     DB1991.DBD  542;
      T     DB1995.DBD  190;
      L     DB1995.DBD  142;
      T     DB1991.DBD  546;

// Write Own Data to CIP
      L     DB1995.DBD   10;
      T     DB1995.DBD  154;

      L     DB1995.DBW   14;
      T     DB1995.DBW  158;

      L     DB1995.DBW   16;
      T     DB1995.DBW  160;

      L     DB1995.DBW   18;
      T     DB1995.DBW  162;

      L     DB1995.DBW   20;
      T     DB1995.DBW  164;

      L     DB1995.DBW   22;
      T     DB1995.DBW  166;

      A     DB1995.DBX   24.0;
      =     DB1995.DBX  168.0;

      A     DB1995.DBX   24.1;
      =     DB1995.DBX  168.1;

      A     DB1995.DBX   24.2;
      =     DB1995.DBX  168.2;

      A     DB1995.DBX   24.3;
      =     DB1995.DBX  168.3;

      A     DB1995.DBX   24.4;
      =     DB1995.DBX  168.4;

      A     DB1995.DBX   24.5;
      =     DB1995.DBX  168.5;

      A     DB1995.DBX   24.6;
      =     DB1995.DBX  168.6;

      A     DB1995.DBX   24.7;
      =     DB1995.DBX  168.7;

// Copy Data to CIP
      CALL SFC   20 (
           SRCBLK                   := DB1995.ToCIP,
           RET_VAL                  := #iRetVal,
           DSTBLK                   := DB1995.ToCIP);

NCIP: NOP   0;

//Empty Signal
//A     "U099SpID".SpI.Sig //!!!! Insert correct Empty Signal !!!
      CLR   ;
      =     DB1995.DBX   26.5;

//Full Signal
//A     "U099SpID".SpI.Sig //!!!! Insert correct Full Signal !!!
      CLR   ;
      =     DB1995.DBX   26.2;

//CIP Program Selected
      A     #CIP;
      =     DB1995.DBX   27.1;

// Emergency Stop
      SET   ;
      =     DB1995.DBX   27.0; //Emergency Stop OK


// Sing bend connections

      A     DB2991.DBX  438.7;
      =     DB1995.DBX   27.2;

      A     DB2991.DBX  498.7;
      =     DB1995.DBX   27.3;


NETWORK
TITLE = read from other unit data






END_FUNCTION_BLOCK

FUNCTION_BLOCK FB 1999
TITLE =U099: PLC 3 General
AUTHOR : Woermann
FAMILY : BOTEC_F1
NAME : Sim
VERSION : 0.1


VAR_TEMP
  CIP : BOOL ;	//CIP active
  xTmp : BOOL ;	//Temporary BOOL (free for general use)
  iTmp : INT ;	//Temporary INT (free for general use)
  rTmp : REAL ;	//Temporary REAL (free for general use)
  UnitNo : INT ;	//Unit Number
END_VAR
BEGIN
NETWORK
TITLE =General

      SET   ;
// get unit number ----------------------------------------------------------
      L     DB1990.DBW    0;
      T     #UnitNo;

// CIP ----------------------------------------------------------------------
      L     DB1991.DBD   54;
      L     0;
      <D    ;
      =     #CIP;

NETWORK
TITLE =Actuator

      A     DB1991.DBX   17.3;
      =     DB2990.DBX  105.3;
      =     DB2990.DBX  185.3;
      =     DB2990.DBX  265.3;

NETWORK
TITLE =Special Input

      A     DB1991.DBX   17.3;
      =     DB2991.DBX   81.3;
      =     DB2991.DBX  141.3;
      =     DB2991.DBX  201.3;
      =     DB2991.DBX  261.3;
      =     DB2991.DBX  321.3;
      =     DB2991.DBX  381.3;
      =     DB2991.DBX  441.3;
      =     DB2991.DBX  501.3;

NETWORK
TITLE =Counter

      A     DB1991.DBX   17.3;
      A     M    101.0;


      CLR   ;
NETWORK
TITLE =Analog Input

      A     DB1991.DBX   17.3;
      =     DB2993.DBX  141.3;

NETWORK
TITLE =Universal Value

      A     DB1991.DBX   17.3;
//      =     "U099UnVD".unv001.Sim;
//      =     "U099UnVD".unv002.Sim;

NETWORK
TITLE =PID

      A     DB1991.DBX   17.3;

NETWORK
TITLE =Message

      A     DB1991.DBX   17.3;
//      =     "U099MsgD".msg001.Sim;
//      =     "U099MsgD".msg002.Sim;

NETWORK
TITLE =VLT

      A     DB1991.DBX   17.3;

END_FUNCTION_BLOCK

FUNCTION_BLOCK FB 4035
TITLE =U103: Transfer Plant 3
FAMILY : BOTEC_F1
NAME : Comm
VERSION : 0.1


VAR_TEMP
  iRetVal : INT ;	//return value as integer
  wRetVal : WORD ;	//return value as word
  Run : BOOL ;	//Unit in "RUN" mode
  EStopOK : BOOL ;	//Emergency Stop OK
  CIP : BOOL ;	//CIP Program Selected
  ComCIP : BOOL ;	//Communication with CIP Active
  xTmp : BOOL ;	//Temporary BOOL (free for general use)
  iTmp : INT ;	//Temporary INT (free for general use)
  rTmp : REAL ;	//Temporary REAL (free for general use)
  dTmp : DINT ;	//Temporary DINT (free for general use)
  UnitNo : INT ;	//Unit Number
  EquipmentID : INT ;	//Equipment ID
  Prid : DINT ;	//Process ID
  SFM36 : STRUCT 	// CIP Pump Mode
   I00 : BOOL ;	// Off
   I01 : BOOL ;	// Flow
   I02 : BOOL ;	// Pressure
   I03 : BOOL ;	// Fix Speed
   I04 : BOOL ;
   I05 : BOOL ;
   I06 : BOOL ;
   I07 : BOOL ;
   I08 : BOOL ;
   I09 : BOOL ;
   I10 : BOOL ;
   I11 : BOOL ;
   I12 : BOOL ;
   I13 : BOOL ;
   I14 : BOOL ;
   I15 : BOOL ;
   I16 : BOOL ;
   I17 : BOOL ;
   I18 : BOOL ;
   I19 : BOOL ;
   I20 : BOOL ;
   I21 : BOOL ;
   I22 : BOOL ;
   I23 : BOOL ;
   I24 : BOOL ;
   I25 : BOOL ;
   I26 : BOOL ;
   I27 : BOOL ;
   I28 : BOOL ;
   I29 : BOOL ;
   I30 : BOOL ;
   I31 : BOOL ;
  END_STRUCT ;
END_VAR
BEGIN
NETWORK
TITLE =general

      SET   ;

// unit & equipment number ---------------------------------------------------
      L     DB4030.DBW    0;
      T     #UnitNo;

      L     DB4035.DBW   14;
      L     1000;
      *I    ;
      L     #UnitNo;
      +I    ;
      T     #EquipmentID;

// CIP ----------------------------------------------------------------------
      L     DB4035.DBW   18;
      L     0;
      <I    ;
      =     #CIP;

// Communicating Units-------------------------------------------------------
      L     DB4035.DBD   10;
      L     DB4035.DBD  106;
      ==D   ;
      =     #ComCIP;

// emergency OK -------------------------------------------------------------
      A     DB4035.DBX   75.0; //General Emergency Stop OK
      =     #EStopOK;

NETWORK
TITLE =remote start

      SET   ;
      A     DB4031.DBX   66.2;
      A     DB4031.DBX   15.0;
      A     DB4031.DBX   17.4;
      JCN   Strt;
      L     DB4035.DBD   10;
      L     L#-1; // Prid negative to start on its own
      T     #Prid;

      CALL FC    48 (
           UnitNo                   := #UnitNo,
           PrId                     := #Prid,
           Run                      := DB4031.DBX   17.4,
           PrIdTransfer             := TRUE,
           Start                    := TRUE,
           RetVal                   := #wRetVal);
Strt: NOP   0;

// Start von Sirupraum (VP3)
      AN    DB1995.DBX 1176.7;
      A     DB1995.DBX 1176.0;
      A     DB4031.DBX   15.0;
      A     DB4031.DBX   17.4;
      JCN   Str2;
      L     DB1995.DBD 1162;
      T     #Prid;

      CALL FC    48 (
           UnitNo                   := #UnitNo,
           PrId                     := #Prid,
           Run                      := DB4031.DBX   17.4,
           PrIdTransfer             := TRUE,
           Start                    := TRUE,
           RetVal                   := #wRetVal);
Str2: NOP   0;

END_FUNCTION_BLOCK

FUNCTION_BLOCK FB 4039
TITLE =U103: Transfer Plant 3
AUTHOR : Woermann
FAMILY : BOTEC_F1
NAME : Sim
VERSION : 0.1


VAR_TEMP
  CIP : BOOL ;	//CIP active
  xTmp : BOOL ;	//Temporary BOOL (free for general use)
  iTmp : INT ;	//Temporary INT (free for general use)
  rTmp : REAL ;	//Temporary REAL (free for general use)
  UnitNo : INT ;	//Unit Number
END_VAR
BEGIN
NETWORK
TITLE =General

      SET   ;
// get unit number ----------------------------------------------------------
      L     DB4030.DBW    0;
      T     #UnitNo;

// CIP ----------------------------------------------------------------------
      L     DB4031.DBD   54;
      L     0;
      <D    ;
      =     #CIP;

NETWORK
TITLE =Actuator

      A     DB4031.DBX   17.3;
      =     DB5030.DBX  425.3;
      =     DB5030.DBX  505.3;
      =     DB5030.DBX  585.3;
      =     DB5030.DBX  665.3;
      =     DB5030.DBX  745.3;
      =     DB5030.DBX  825.3;
      =     DB5030.DBX  905.3;
      =     DB5030.DBX  985.3;
      =     DB5030.DBX 1065.3;
      =     DB5030.DBX 1145.3;
      =     DB5030.DBX 1225.3;
      =     DB5030.DBX 1305.3;
      =     DB5030.DBX 2665.3;
      =     DB5030.DBX 2745.3;
      =     DB5030.DBX 2825.3;
      =     DB5030.DBX 2905.3;
      =     DB5030.DBX 3065.3;
      =     DB5030.DBX 3145.3;
      =     DB5030.DBX 3225.3;
      =     DB5030.DBX 3305.3;

NETWORK
TITLE =Special Input

      A     DB4031.DBX   17.3;
      =     DB5031.DBX  681.3;
      =     DB5031.DBX  741.3;
      =     DB5031.DBX 1041.3;
      =     DB5031.DBX 1101.3;
      =     DB5031.DBX 1221.3;
      =     DB5031.DBX 1281.3;
      =     DB5031.DBX 1341.3;
      =     DB5031.DBX 1761.3;
      =     DB5031.DBX 1881.3;
      =     DB5031.DBX 1941.3;


NETWORK
TITLE =Counter

      A     DB4031.DBX   17.3;
      A     M    101.0;


      CLR   ;
NETWORK
TITLE =Analog Input

      A     DB4031.DBX   17.3;

NETWORK
TITLE =Universal Value

      A     DB4031.DBX   17.3;
//      =     "U103UnVD".unv001.Sim;
//      =     "U103UnVD".unv002.Sim;
//      =     "U103UnVD".unv003.Sim;
//      =     "U103UnVD".unv004.Sim;

NETWORK
TITLE =PID

      A     DB4031.DBX   17.3;

NETWORK
TITLE =Message

      A     DB4031.DBX   17.3;
//      =     "U103MsgD".msg001.Sim;
//      =     "U103MsgD".msg002.Sim;
//      =     "U103MsgD".msg003.Sim;

NETWORK
TITLE =VLT

      A     DB4031.DBX   17.3;

END_FUNCTION_BLOCK

FUNCTION_BLOCK FB 4055
TITLE =U105: Transfer Plant 5
FAMILY : BOTEC_F1
NAME : Comm
VERSION : 0.1


VAR_TEMP
  iRetVal : INT ;	//return value as integer
  wRetVal : WORD ;	//return value as word
  Run : BOOL ;	//Unit in "RUN" mode
  EStopOK : BOOL ;	//Emergency Stop OK
  CIP : BOOL ;	//CIP Program Selected
  ComCIP : BOOL ;	//Communication with CIP Active
  xTmp : BOOL ;	//Temporary BOOL (free for general use)
  iTmp : INT ;	//Temporary INT (free for general use)
  rTmp : REAL ;	//Temporary REAL (free for general use)
  dTmp : DINT ;	//Temporary DINT (free for general use)
  UnitNo : INT ;	//Unit Number
  EquipmentID : INT ;	//Equipment ID
  Prid : DINT ;	//Process ID
  SFM36 : STRUCT 	// CIP Pump Mode
   I00 : BOOL ;	// Off
   I01 : BOOL ;	// Flow
   I02 : BOOL ;	// Pressure
   I03 : BOOL ;	// Fix Speed
   I04 : BOOL ;
   I05 : BOOL ;
   I06 : BOOL ;
   I07 : BOOL ;
   I08 : BOOL ;
   I09 : BOOL ;
   I10 : BOOL ;
   I11 : BOOL ;
   I12 : BOOL ;
   I13 : BOOL ;
   I14 : BOOL ;
   I15 : BOOL ;
   I16 : BOOL ;
   I17 : BOOL ;
   I18 : BOOL ;
   I19 : BOOL ;
   I20 : BOOL ;
   I21 : BOOL ;
   I22 : BOOL ;
   I23 : BOOL ;
   I24 : BOOL ;
   I25 : BOOL ;
   I26 : BOOL ;
   I27 : BOOL ;
   I28 : BOOL ;
   I29 : BOOL ;
   I30 : BOOL ;
   I31 : BOOL ;
  END_STRUCT ;
END_VAR
BEGIN
NETWORK
TITLE =general

      SET   ;

// unit & equipment number ---------------------------------------------------
      L     DB4050.DBW    0;
      T     #UnitNo;

      L     DB4055.DBW   14;
      L     1000;
      *I    ;
      L     #UnitNo;
      +I    ;
      T     #EquipmentID;

// CIP ----------------------------------------------------------------------
      L     DB4055.DBW   18;
      L     0;
      <I    ;
      =     #CIP;

// Communicating Units-------------------------------------------------------
      L     DB4055.DBD   10;
      L     DB4055.DBD  106;
      ==D   ;
      =     #ComCIP;

// emergency OK -------------------------------------------------------------
      A     DB4055.DBX   75.0; //General Emergency Stop OK
      =     #EStopOK;

NETWORK
TITLE =remote start

      SET   ;
      A     DB4051.DBX   66.2;
      A     DB4051.DBX   15.0;
      A     DB4051.DBX   17.4;
      JCN   Strt;
      L     DB4055.DBD   10;
      L     L#-1; // Prid negative to start on its own
      T     #Prid;

      CALL FC    48 (
           UnitNo                   := #UnitNo,
           PrId                     := #Prid,
           Run                      := DB4051.DBX   17.4,
           PrIdTransfer             := TRUE,
           Start                    := TRUE,
           RetVal                   := #wRetVal);
Strt: NOP   0;

// Start von Sirupraum (VP3)
      AN    DB1995.DBX 1224.7;
      A     DB1995.DBX 1224.0;
      A     DB4051.DBX   15.0;
      A     DB4051.DBX   17.4;
      JCN   Str2;
      L     DB1995.DBD 1210;
      T     #Prid;

      CALL FC    48 (
           UnitNo                   := #UnitNo,
           PrId                     := #Prid,
           Run                      := DB4051.DBX   17.4,
           PrIdTransfer             := TRUE,
           Start                    := TRUE,
           RetVal                   := #wRetVal);
Str2: NOP   0;

END_FUNCTION_BLOCK

FUNCTION_BLOCK FB 4059
TITLE =U105: Transfer Plant 5
AUTHOR : Woermann
FAMILY : BOTEC_F1
NAME : Sim
VERSION : 0.1


VAR_TEMP
  CIP : BOOL ;	//CIP active
  xTmp : BOOL ;	//Temporary BOOL (free for general use)
  iTmp : INT ;	//Temporary INT (free for general use)
  rTmp : REAL ;	//Temporary REAL (free for general use)
  UnitNo : INT ;	//Unit Number
END_VAR
BEGIN
NETWORK
TITLE =General

      SET   ;
// get unit number ----------------------------------------------------------
      L     DB4050.DBW    0;
      T     #UnitNo;

// CIP ----------------------------------------------------------------------
      L     DB4051.DBD   54;
      L     0;
      <D    ;
      =     #CIP;

NETWORK
TITLE =Actuator

      A     DB4051.DBX   17.3;
      =     DB5050.DBX  105.3;
      =     DB5050.DBX  185.3;
      =     DB5050.DBX  265.3;
      =     DB5050.DBX  345.3;
      =     DB5050.DBX  425.3;
      =     DB5050.DBX  505.3;
      =     DB5050.DBX  585.3;
      =     DB5050.DBX  665.3;
      =     DB5050.DBX  745.3;
      =     DB5050.DBX  825.3;
      =     DB5050.DBX  905.3;
      =     DB5050.DBX  985.3;
      =     DB5050.DBX 1065.3;
      =     DB5050.DBX 1145.3;
      =     DB5050.DBX 1225.3;
      =     DB5050.DBX 1305.3;
      =     DB5050.DBX 1385.3;
      =     DB5050.DBX 1465.3;
      =     DB5050.DBX 1545.3;
      =     DB5050.DBX 1625.3;
      =     DB5050.DBX 1705.3;
      =     DB5050.DBX 1785.3;
      =     DB5050.DBX 1865.3;
      =     DB5050.DBX 2345.3;
      =     DB5050.DBX 3065.3;
      =     DB5050.DBX 3145.3;
      =     DB5050.DBX 3225.3;
      =     DB5050.DBX 3305.3;

NETWORK
TITLE =Special Input

      A     DB4051.DBX   17.3;
      =     DB5051.DBX   81.3;
      =     DB5051.DBX  141.3;
      =     DB5051.DBX  201.3;
      =     DB5051.DBX  261.3;
      =     DB5051.DBX  321.3;
      =     DB5051.DBX  381.3;
      =     DB5051.DBX  441.3;
      =     DB5051.DBX  501.3;
      =     DB5051.DBX  561.3;
      =     DB5051.DBX  621.3;
      =     DB5051.DBX  681.3;
      =     DB5051.DBX  741.3;
      =     DB5051.DBX  801.3;
      =     DB5051.DBX 1041.3;
      =     DB5051.DBX 1101.3;
      =     DB5051.DBX 1161.3;
      =     DB5051.DBX 1221.3;
      =     DB5051.DBX 1281.3;
      =     DB5051.DBX 1341.3;
      =     DB5051.DBX 1461.3;
      =     DB5051.DBX 1521.3;
      =     DB5051.DBX 1581.3;
      =     DB5051.DBX 1641.3;
      =     DB5051.DBX 1701.3;
      =     DB5051.DBX 1761.3;
      =     DB5051.DBX 1821.3;
      =     DB5051.DBX 1881.3;
      =     DB5051.DBX 1941.3;
      =     DB5051.DBX 2001.3;
      =     DB5051.DBX 2061.3;


NETWORK
TITLE =Counter

      A     DB4051.DBX   17.3;
      A     M    101.0;


      CLR   ;
NETWORK
TITLE =Analog Input

      A     DB4051.DBX   17.3;
      =     DB5053.DBX  141.3;

NETWORK
TITLE =Universal Value

      A     DB4051.DBX   17.3;
//      =     "U105UnVD".unv001.Sim;
//      =     "U105UnVD".unv002.Sim;
//      =     "U105UnVD".unv003.Sim;
//      =     "U105UnVD".unv004.Sim;

NETWORK
TITLE =PID

      A     DB4051.DBX   17.3;

NETWORK
TITLE =Message

      A     DB4051.DBX   17.3;
//      =     "U105MsgD".msg001.Sim;
//      =     "U105MsgD".msg002.Sim;
//      =     "U105MsgD".msg003.Sim;

NETWORK
TITLE =VLT

      A     DB4051.DBX   17.3;

END_FUNCTION_BLOCK

FUNCTION_BLOCK FB 4075
TITLE =U107: Transfer Plant 7
FAMILY : BOTEC_F1
NAME : Comm
VERSION : 0.1


VAR_TEMP
  iRetVal : INT ;	//return value as integer
  wRetVal : WORD ;	//return value as word
  Run : BOOL ;	//Unit in "RUN" mode
  EStopOK : BOOL ;	//Emergency Stop OK
  CIP : BOOL ;	//CIP Program Selected
  ComCIP : BOOL ;	//Communication with CIP Active
  xTmp : BOOL ;	//Temporary BOOL (free for general use)
  iTmp : INT ;	//Temporary INT (free for general use)
  rTmp : REAL ;	//Temporary REAL (free for general use)
  dTmp : DINT ;	//Temporary DINT (free for general use)
  UnitNo : INT ;	//Unit Number
  EquipmentID : INT ;	//Equipment ID
  Prid : DINT ;	//Process ID
  SFM36 : STRUCT 	// CIP Pump Mode
   I00 : BOOL ;	// Off
   I01 : BOOL ;	// Flow
   I02 : BOOL ;	// Pressure
   I03 : BOOL ;	// Fix Speed
   I04 : BOOL ;
   I05 : BOOL ;
   I06 : BOOL ;
   I07 : BOOL ;
   I08 : BOOL ;
   I09 : BOOL ;
   I10 : BOOL ;
   I11 : BOOL ;
   I12 : BOOL ;
   I13 : BOOL ;
   I14 : BOOL ;
   I15 : BOOL ;
   I16 : BOOL ;
   I17 : BOOL ;
   I18 : BOOL ;
   I19 : BOOL ;
   I20 : BOOL ;
   I21 : BOOL ;
   I22 : BOOL ;
   I23 : BOOL ;
   I24 : BOOL ;
   I25 : BOOL ;
   I26 : BOOL ;
   I27 : BOOL ;
   I28 : BOOL ;
   I29 : BOOL ;
   I30 : BOOL ;
   I31 : BOOL ;
  END_STRUCT ;
END_VAR
BEGIN
NETWORK
TITLE =general

      SET   ;

// unit & equipment number ---------------------------------------------------
      L     DB4070.DBW    0;
      T     #UnitNo;

      L     DB4075.DBW   14;
      L     1000;
      *I    ;
      L     #UnitNo;
      +I    ;
      T     #EquipmentID;

// CIP ----------------------------------------------------------------------
      L     DB4075.DBW   18;
      L     0;
      <I    ;
      =     #CIP;

// Communicating Units-------------------------------------------------------
      L     DB4075.DBD   10;
      L     DB4075.DBD  106;
      ==D   ;
      =     #ComCIP;

// emergency OK -------------------------------------------------------------
      A     DB4075.DBX   75.0; //General Emergency Stop OK
      =     #EStopOK;

NETWORK
TITLE =remote start

      SET   ;
      A     DB4071.DBX   66.2;
      A     DB4071.DBX   15.0;
      A     DB4071.DBX   17.4;
      JCN   Strt;
      L     DB4075.DBD   10;
      L     L#-1; // Prid negative to start on its own
      T     #Prid;

      CALL FC    48 (
           UnitNo                   := #UnitNo,
           PrId                     := #Prid,
           Run                      := DB4071.DBX   17.4,
           PrIdTransfer             := TRUE,
           Start                    := TRUE,
           RetVal                   := #wRetVal);
Strt: NOP   0;

// Start von Sirupraum (VP3)
      AN    DB1995.DBX 1272.7;
      A     DB1995.DBX 1272.0;
      A     DB4071.DBX   15.0;
      A     DB4071.DBX   17.4;
      JCN   Str2;
      L     DB1995.DBD 1258;
      T     #Prid;

      CALL FC    48 (
           UnitNo                   := #UnitNo,
           PrId                     := #Prid,
           Run                      := DB4071.DBX   17.4,
           PrIdTransfer             := TRUE,
           Start                    := TRUE,
           RetVal                   := #wRetVal);
Str2: NOP   0;

END_FUNCTION_BLOCK

FUNCTION_BLOCK FB 4079
TITLE =U107: Transfer Plant 7
AUTHOR : Woermann
FAMILY : BOTEC_F1
NAME : Sim
VERSION : 0.1


VAR_TEMP
  CIP : BOOL ;	//CIP active
  xTmp : BOOL ;	//Temporary BOOL (free for general use)
  iTmp : INT ;	//Temporary INT (free for general use)
  rTmp : REAL ;	//Temporary REAL (free for general use)
  UnitNo : INT ;	//Unit Number
END_VAR
BEGIN
NETWORK
TITLE =General

      SET   ;
// get unit number ----------------------------------------------------------
      L     DB4070.DBW    0;
      T     #UnitNo;

// CIP ----------------------------------------------------------------------
      L     DB4071.DBD   54;
      L     0;
      <D    ;
      =     #CIP;

NETWORK
TITLE =Actuator

      A     DB4071.DBX   17.3;
      =     DB5070.DBX  425.3;
      =     DB5070.DBX  505.3;
      =     DB5070.DBX  585.3;
      =     DB5070.DBX  665.3;
      =     DB5070.DBX  745.3;
      =     DB5070.DBX  825.3;
      =     DB5070.DBX  905.3;
      =     DB5070.DBX  985.3;
      =     DB5070.DBX 1065.3;
      =     DB5070.DBX 1145.3;
      =     DB5070.DBX 1225.3;
      =     DB5070.DBX 1305.3;
      =     DB5070.DBX 1385.3;
      =     DB5070.DBX 1465.3;
      =     DB5070.DBX 1945.3;
      =     DB5070.DBX 2025.3;
      =     DB5070.DBX 2105.3;
      =     DB5070.DBX 2185.3;
      =     DB5070.DBX 2265.3;
      =     DB5070.DBX 2345.3;
      =     DB5070.DBX 2425.3;
      =     DB5070.DBX 2505.3;
      =     DB5070.DBX 2585.3;
      =     DB5070.DBX 2665.3;
      =     DB5070.DBX 2745.3;
      =     DB5070.DBX 2825.3;
      =     DB5070.DBX 2905.3;
      =     DB5070.DBX 2985.3;
      =     DB5070.DBX 3065.3;
      =     DB5070.DBX 3145.3;
      =     DB5070.DBX 3225.3;
      =     DB5070.DBX 3305.3;

NETWORK
TITLE =Special Input

      A     DB4071.DBX   17.3;
      =     DB5071.DBX  681.3;
      =     DB5071.DBX  741.3;
      =     DB5071.DBX 1041.3;
      =     DB5071.DBX 1101.3;
      =     DB5071.DBX 1161.3;
      =     DB5071.DBX 1221.3;
      =     DB5071.DBX 1281.3;
      =     DB5071.DBX 1341.3;
      =     DB5071.DBX 1461.3;
      =     DB5071.DBX 1521.3;
      =     DB5071.DBX 1581.3;
      =     DB5071.DBX 1761.3;
      =     DB5071.DBX 1821.3;
      =     DB5071.DBX 1881.3;
      =     DB5071.DBX 1941.3;
      =     DB5071.DBX 2001.3;
      =     DB5071.DBX 2061.3;

NETWORK
TITLE =Counter

      A     DB4071.DBX   17.3;
      A     M    101.0;


      CLR   ;
NETWORK
TITLE =Analog Input

      A     DB4071.DBX   17.3;

NETWORK
TITLE =Universal Value

      A     DB4071.DBX   17.3;
//      =     "U107UnVD".unv001.Sim;
//      =     "U107UnVD".unv002.Sim;
//      =     "U107UnVD".unv003.Sim;
//      =     "U107UnVD".unv004.Sim;

NETWORK
TITLE =PID

      A     DB4071.DBX   17.3;

NETWORK
TITLE =Message

      A     DB4071.DBX   17.3;
//      =     "U107MsgD".msg001.Sim;
//      =     "U107MsgD".msg002.Sim;
//      =     "U107MsgD".msg003.Sim;

NETWORK
TITLE =VLT

      A     DB4071.DBX   17.3;

END_FUNCTION_BLOCK

FUNCTION_BLOCK FB 4085
TITLE =U108: Transfer Plant 8
FAMILY : BOTEC_F1
NAME : Comm
VERSION : 0.1


VAR_TEMP
  iRetVal : INT ;	//return value as integer
  wRetVal : WORD ;	//return value as word
  Run : BOOL ;	//Unit in "RUN" mode
  EStopOK : BOOL ;	//Emergency Stop OK
  CIP : BOOL ;	//CIP Program Selected
  ComCIP : BOOL ;	//Communication with CIP Active
  xTmp : BOOL ;	//Temporary BOOL (free for general use)
  iTmp : INT ;	//Temporary INT (free for general use)
  rTmp : REAL ;	//Temporary REAL (free for general use)
  dTmp : DINT ;	//Temporary DINT (free for general use)
  UnitNo : INT ;	//Unit Number
  EquipmentID : INT ;	//Equipment ID
  Prid : DINT ;	//Process ID
  SFM36 : STRUCT 	// CIP Pump Mode
   I00 : BOOL ;	// Off
   I01 : BOOL ;	// Flow
   I02 : BOOL ;	// Pressure
   I03 : BOOL ;	// Fix Speed
   I04 : BOOL ;
   I05 : BOOL ;
   I06 : BOOL ;
   I07 : BOOL ;
   I08 : BOOL ;
   I09 : BOOL ;
   I10 : BOOL ;
   I11 : BOOL ;
   I12 : BOOL ;
   I13 : BOOL ;
   I14 : BOOL ;
   I15 : BOOL ;
   I16 : BOOL ;
   I17 : BOOL ;
   I18 : BOOL ;
   I19 : BOOL ;
   I20 : BOOL ;
   I21 : BOOL ;
   I22 : BOOL ;
   I23 : BOOL ;
   I24 : BOOL ;
   I25 : BOOL ;
   I26 : BOOL ;
   I27 : BOOL ;
   I28 : BOOL ;
   I29 : BOOL ;
   I30 : BOOL ;
   I31 : BOOL ;
  END_STRUCT ;
END_VAR
BEGIN
NETWORK
TITLE =general

      SET   ;

// unit & equipment number ---------------------------------------------------
      L     DB4080.DBW    0;
      T     #UnitNo;

      L     DB4085.DBW   14;
      L     1000;
      *I    ;
      L     #UnitNo;
      +I    ;
      T     #EquipmentID;

// CIP ----------------------------------------------------------------------
      L     DB4085.DBW   18;
      L     0;
      <I    ;
      =     #CIP;

// Communicating Units-------------------------------------------------------
      L     DB4085.DBD   10;
      L     DB4085.DBD  106;
      ==D   ;
      =     #ComCIP;

// emergency OK -------------------------------------------------------------
      A     DB4085.DBX   75.0; //General Emergency Stop OK
      =     #EStopOK;

NETWORK
TITLE =read other unit's data

      SET   ;

// ... General Unit ----------/

      CALL FC   563 (
           ActReq                   := M    101.0,
           PLCNo                    := DB4085.DBW   14,
           SourceUnitNo             := 99,
           IsTUnit                  := FALSE,
           DstComDRec               := DB4085.GEN,
           RET_VAL                  := #wRetVal);

NETWORK
TITLE =remote start

      SET   ;
      A     DB4081.DBX   66.2;
//      O     DB5081.DBX 1098.7
      A     DB4081.DBX   15.0;
      A     DB4081.DBX   17.4;
      CLR   ;
      JCN   Strt;
      L     L#-1; // Prid negative to start on its own
      T     #Prid;

      CALL FC    48 (
           UnitNo                   := #UnitNo,
           PrId                     := #Prid,
           Run                      := DB4081.DBX   17.4,
           PrIdTransfer             := TRUE,
           Start                    := TRUE,
           RetVal                   := #wRetVal);
Strt: NOP   0;
NETWORK
TITLE =external releases

      SET   ;

NETWORK
TITLE =write own unit data

      SET   ;

//-- CIP Communication ---------------------------------------
      AN    DB4081.DBX   15.0;
//      AN "U108SeqD".Seq.PO.B30 // CIP Active (Slave)
      A     #ComCIP;
      JCN   NCIP;
//Conductivity CIP Return
      L     DB4085.DBD  150;
      T     DB4081.DBD  626;

//Temperature CIP Return
      L     DB4085.DBD  146;
      T     DB4081.DBD  594;

//CIP Prerun Pump SP

      CALL FC    45 (
           SFM                      := DB4081.DBD  686,
           Indexes                  := #SFM36);


      L     0.000000e+000;
      A     #SFM36.I01;
      =     DB4085.DBX  171.7;
      JCN   pfc;
      L     DB4081.DBD  654;
pfc:  NOP   0;
      A     #SFM36.I02;
      =     DB4085.DBX  172.0;
      JCN   ppc;
      L     DB4081.DBD  670;
ppc:  NOP   0;
      A     #SFM36.I03;
      =     DB4085.DBX  171.6;
      JCN   pxc;
      L     DB4081.DBD  574;
pxc:  NOP   0;
      T     DB4085.DBD  182;

//CIP Return
      L     DB4081.DBD  558;
      T     DB4085.DBD  186;
      L     DB4085.DBD  138;
      T     DB4081.DBD  562;

//CIP Prerun
      L     DB4081.DBD  542;
      T     DB4085.DBD  190;
      L     DB4085.DBD  142;
      T     DB4081.DBD  546;

// Write Own Data to CIP
      L     DB4085.DBD   10;
      T     DB4085.DBD  154;

      L     DB4085.DBW   14;
      T     DB4085.DBW  158;

      L     DB4085.DBW   16;
      T     DB4085.DBW  160;

      L     DB4085.DBW   18;
      T     DB4085.DBW  162;

      L     DB4085.DBW   20;
      T     DB4085.DBW  164;

      L     DB4085.DBW   22;
      T     DB4085.DBW  166;

      A     DB4085.DBX   24.0;
      =     DB4085.DBX  168.0;

      A     DB4085.DBX   24.1;
      =     DB4085.DBX  168.1;

      A     DB4085.DBX   24.2;
      =     DB4085.DBX  168.2;

      A     DB4085.DBX   24.3;
      =     DB4085.DBX  168.3;

      A     DB4085.DBX   24.4;
      =     DB4085.DBX  168.4;

      A     DB4085.DBX   24.5;
      =     DB4085.DBX  168.5;

      A     DB4085.DBX   24.6;
      =     DB4085.DBX  168.6;

      A     DB4085.DBX   24.7;
      =     DB4085.DBX  168.7;

// Copy Data to CIP
      CALL SFC   20 (
           SRCBLK                   := DB4085.ToCIP,
           RET_VAL                  := #iRetVal,
           DSTBLK                   := DB4085.ToCIP);

NCIP: NOP   0;

//Empty Signal
//A     "U108SpID".SpI.Sig //!!!! Insert correct Empty Signal !!!
      CLR   ;
      =     DB4085.DBX   26.5;

//Full Signal
//A     "U108SpID".SpI.Sig //!!!! Insert correct Full Signal !!!
      CLR   ;
      =     DB4085.DBX   26.2;

//CIP Program Selected
      A     #CIP;
      =     DB4085.DBX   27.1;

// Emergency Stop
      A     #EStopOK; //If needed add or replace with own SpI
      =     DB4085.DBX   27.0; //Emergency Stop OK


NETWORK
TITLE = read from other unit data



END_FUNCTION_BLOCK

FUNCTION_BLOCK FB 4089
TITLE =U108: Transfer Plant 8
AUTHOR : Woermann
FAMILY : BOTEC_F1
NAME : Sim
VERSION : 0.1


VAR_TEMP
  CIP : BOOL ;	//CIP active
  xTmp : BOOL ;	//Temporary BOOL (free for general use)
  iTmp : INT ;	//Temporary INT (free for general use)
  rTmp : REAL ;	//Temporary REAL (free for general use)
  UnitNo : INT ;	//Unit Number
END_VAR
BEGIN
NETWORK
TITLE =General

      SET   ;
// get unit number ----------------------------------------------------------
      L     DB4080.DBW    0;
      T     #UnitNo;

// CIP ----------------------------------------------------------------------
      L     DB4081.DBD   54;
      L     0;
      <D    ;
      =     #CIP;

NETWORK
TITLE =Actuator

      A     DB4081.DBX   17.3;

NETWORK
TITLE =Special Input

      A     DB4081.DBX   17.3;

NETWORK
TITLE =Counter

      A     DB4081.DBX   17.3;
      A     M    101.0;


      CLR   ;
NETWORK
TITLE =Analog Input

      A     DB4081.DBX   17.3;

NETWORK
TITLE =Universal Value

      A     DB4081.DBX   17.3;
//      =     "U108UnVD".unv001.Sim;
//      =     "U108UnVD".unv002.Sim;
//      =     "U108UnVD".unv003.Sim;
//      =     "U108UnVD".unv004.Sim;

NETWORK
TITLE =PID

      A     DB4081.DBX   17.3;

NETWORK
TITLE =Message

      A     DB4081.DBX   17.3;
//      =     "U108MsgD".msg001.Sim;
//      =     "U108MsgD".msg002.Sim;
//      =     "U108MsgD".msg003.Sim;

NETWORK
TITLE =VLT

      A     DB4081.DBX   17.3;

END_FUNCTION_BLOCK

FUNCTION_BLOCK FB 4095
TITLE =U109: Transfer Plant 9
FAMILY : BOTEC_F1
NAME : Comm
VERSION : 0.1


VAR_TEMP
  iRetVal : INT ;	//return value as integer
  wRetVal : WORD ;	//return value as word
  Run : BOOL ;	//Unit in "RUN" mode
  EStopOK : BOOL ;	//Emergency Stop OK
  CIP : BOOL ;	//CIP Program Selected
  ComCIP : BOOL ;	//Communication with CIP Active
  xTmp : BOOL ;	//Temporary BOOL (free for general use)
  iTmp : INT ;	//Temporary INT (free for general use)
  rTmp : REAL ;	//Temporary REAL (free for general use)
  dTmp : DINT ;	//Temporary DINT (free for general use)
  UnitNo : INT ;	//Unit Number
  EquipmentID : INT ;	//Equipment ID
  Prid : DINT ;	//Process ID
  SFM36 : STRUCT 	// CIP Pump Mode
   I00 : BOOL ;	// Off
   I01 : BOOL ;	// Flow
   I02 : BOOL ;	// Pressure
   I03 : BOOL ;	// Fix Speed
   I04 : BOOL ;
   I05 : BOOL ;
   I06 : BOOL ;
   I07 : BOOL ;
   I08 : BOOL ;
   I09 : BOOL ;
   I10 : BOOL ;
   I11 : BOOL ;
   I12 : BOOL ;
   I13 : BOOL ;
   I14 : BOOL ;
   I15 : BOOL ;
   I16 : BOOL ;
   I17 : BOOL ;
   I18 : BOOL ;
   I19 : BOOL ;
   I20 : BOOL ;
   I21 : BOOL ;
   I22 : BOOL ;
   I23 : BOOL ;
   I24 : BOOL ;
   I25 : BOOL ;
   I26 : BOOL ;
   I27 : BOOL ;
   I28 : BOOL ;
   I29 : BOOL ;
   I30 : BOOL ;
   I31 : BOOL ;
  END_STRUCT ;
END_VAR
BEGIN
NETWORK
TITLE =general

      SET   ;

// unit & equipment number ---------------------------------------------------
      L     DB4090.DBW    0;
      T     #UnitNo;

      L     DB4095.DBW   14;
      L     1000;
      *I    ;
      L     #UnitNo;
      +I    ;
      T     #EquipmentID;

// CIP ----------------------------------------------------------------------
      L     DB4095.DBW   18;
      L     0;
      <I    ;
      =     #CIP;

// Communicating Units-------------------------------------------------------
      L     DB4095.DBD   10;
      L     DB4095.DBD  106;
      ==D   ;
      =     #ComCIP;

// emergency OK -------------------------------------------------------------
      A     DB4095.DBX   75.0; //General Emergency Stop OK
      =     #EStopOK;

NETWORK
TITLE =remote start

      SET   ;
      A     DB4091.DBX   66.2;
      A     DB4091.DBX   15.0;
      A     DB4091.DBX   17.4;
      JCN   Strt;
      L     DB4095.DBD   10;
      L     L#-1; // Prid negative to start on its own
      T     #Prid;

      CALL FC    48 (
           UnitNo                   := #UnitNo,
           PrId                     := #Prid,
           Run                      := DB4091.DBX   17.4,
           PrIdTransfer             := TRUE,
           Start                    := TRUE,
           RetVal                   := #wRetVal);
Strt: NOP   0;

// Start von Sirupraum (VP3)
      AN    DB1995.DBX 1320.7;
      A     DB1995.DBX 1320.0;
      A     DB4091.DBX   15.0;
      A     DB4091.DBX   17.4;
      JCN   Str2;
      L     DB1995.DBD 1306;
      T     #Prid;

      CALL FC    48 (
           UnitNo                   := #UnitNo,
           PrId                     := #Prid,
           Run                      := DB4091.DBX   17.4,
           PrIdTransfer             := TRUE,
           Start                    := TRUE,
           RetVal                   := #wRetVal);
Str2: NOP   0;


END_FUNCTION_BLOCK

FUNCTION_BLOCK FB 4099
TITLE =U109: Transfer Plant 9
AUTHOR : Woermann
FAMILY : BOTEC_F1
NAME : Sim
VERSION : 0.1


VAR_TEMP
  CIP : BOOL ;	//CIP active
  xTmp : BOOL ;	//Temporary BOOL (free for general use)
  iTmp : INT ;	//Temporary INT (free for general use)
  rTmp : REAL ;	//Temporary REAL (free for general use)
  UnitNo : INT ;	//Unit Number
END_VAR
BEGIN
NETWORK
TITLE =General

      SET   ;
// get unit number ----------------------------------------------------------
      L     DB4090.DBW    0;
      T     #UnitNo;

// CIP ----------------------------------------------------------------------
      L     DB4091.DBD   54;
      L     0;
      <D    ;
      =     #CIP;

NETWORK
TITLE =Actuator

      A     DB4091.DBX   17.3;
      =     DB5090.DBX  425.3;
      =     DB5090.DBX  505.3;
      =     DB5090.DBX  585.3;
      =     DB5090.DBX  665.3;
      =     DB5090.DBX  745.3;
      =     DB5090.DBX  825.3;
      =     DB5090.DBX  905.3;
      =     DB5090.DBX  985.3;
      =     DB5090.DBX 1065.3;
      =     DB5090.DBX 1145.3;
      =     DB5090.DBX 1225.3;
      =     DB5090.DBX 1305.3;
      =     DB5090.DBX 1385.3;
      =     DB5090.DBX 3065.3;
      =     DB5090.DBX 3145.3;
      =     DB5090.DBX 3225.3;
      =     DB5090.DBX 3305.3;


NETWORK
TITLE =Special Input

      A     DB4091.DBX   17.3;
      =     DB5091.DBX   81.3;
      =     DB5091.DBX  681.3;
      =     DB5091.DBX  741.3;
      =     DB5091.DBX 1041.3;
      =     DB5091.DBX 1101.3;
      =     DB5091.DBX 1161.3;
      =     DB5091.DBX 1221.3;
      =     DB5091.DBX 1281.3;
      =     DB5091.DBX 1341.3;
      =     DB5091.DBX 1461.3;
      =     DB5091.DBX 1521.3;
      =     DB5091.DBX 1581.3;
      =     DB5091.DBX 1641.3;
      =     DB5091.DBX 1701.3;
      =     DB5091.DBX 1761.3;
      =     DB5091.DBX 2001.3;
      =     DB5091.DBX 2061.3;

NETWORK
TITLE =Counter

      A     DB4091.DBX   17.3;
      A     M    101.0;


      CLR   ;
NETWORK
TITLE =Analog Input

      A     DB4091.DBX   17.3;

NETWORK
TITLE =Universal Value

      A     DB4091.DBX   17.3;
//      =     "U109UnVD".unv001.Sim;
//      =     "U109UnVD".unv002.Sim;
//      =     "U109UnVD".unv003.Sim;
//      =     "U109UnVD".unv004.Sim;

NETWORK
TITLE =PID

      A     DB4091.DBX   17.3;

NETWORK
TITLE =Message

      A     DB4091.DBX   17.3;
//      =     "U109MsgD".msg001.Sim;
//      =     "U109MsgD".msg002.Sim;
//      =     "U109MsgD".msg003.Sim;

NETWORK
TITLE =VLT

      A     DB4091.DBX   17.3;

END_FUNCTION_BLOCK

FUNCTION_BLOCK FB 4115
TITLE =U111: Transfer Plant 11
FAMILY : BOTEC_F1
NAME : Comm
VERSION : 0.1


VAR_TEMP
  iRetVal : INT ;	//return value as integer
  wRetVal : WORD ;	//return value as word
  Run : BOOL ;	//Unit in "RUN" mode
  EStopOK : BOOL ;	//Emergency Stop OK
  CIP : BOOL ;	//CIP Program Selected
  ComCIP : BOOL ;	//Communication with CIP Active
  xTmp : BOOL ;	//Temporary BOOL (free for general use)
  iTmp : INT ;	//Temporary INT (free for general use)
  rTmp : REAL ;	//Temporary REAL (free for general use)
  dTmp : DINT ;	//Temporary DINT (free for general use)
  UnitNo : INT ;	//Unit Number
  EquipmentID : INT ;	//Equipment ID
  Prid : DINT ;	//Process ID
  SFM36 : STRUCT 	// CIP Pump Mode
   I00 : BOOL ;	// Off
   I01 : BOOL ;	// Flow
   I02 : BOOL ;	// Pressure
   I03 : BOOL ;	// Fix Speed
   I04 : BOOL ;
   I05 : BOOL ;
   I06 : BOOL ;
   I07 : BOOL ;
   I08 : BOOL ;
   I09 : BOOL ;
   I10 : BOOL ;
   I11 : BOOL ;
   I12 : BOOL ;
   I13 : BOOL ;
   I14 : BOOL ;
   I15 : BOOL ;
   I16 : BOOL ;
   I17 : BOOL ;
   I18 : BOOL ;
   I19 : BOOL ;
   I20 : BOOL ;
   I21 : BOOL ;
   I22 : BOOL ;
   I23 : BOOL ;
   I24 : BOOL ;
   I25 : BOOL ;
   I26 : BOOL ;
   I27 : BOOL ;
   I28 : BOOL ;
   I29 : BOOL ;
   I30 : BOOL ;
   I31 : BOOL ;
  END_STRUCT ;
END_VAR
BEGIN
NETWORK
TITLE =general

      SET   ;

// unit & equipment number ---------------------------------------------------
      L     DB4110.DBW    0;
      T     #UnitNo;

      L     DB4115.DBW   14;
      L     1000;
      *I    ;
      L     #UnitNo;
      +I    ;
      T     #EquipmentID;

// CIP ----------------------------------------------------------------------
      L     DB4115.DBW   18;
      L     0;
      <I    ;
      =     #CIP;

// Communicating Units-------------------------------------------------------
      L     DB4115.DBD   10;
      L     DB4115.DBD  106;
      ==D   ;
      =     #ComCIP;

// emergency OK -------------------------------------------------------------
      A     DB4115.DBX   75.0; //General Emergency Stop OK
      =     #EStopOK;

NETWORK
TITLE =remote start

      SET   ;
      A     DB4111.DBX   66.2;
      O     DB5111.DBX 1098.7;
      A     DB4111.DBX   15.0;
      A     DB4111.DBX   17.4;
      CLR   ;
      JCN   Strt;
      L     DB4115.DBD   10;
      L     L#-1; // Prid negative to start on its own
      T     #Prid;

      CALL FC    48 (
           UnitNo                   := #UnitNo,
           PrId                     := #Prid,
           Run                      := DB4111.DBX   17.4,
           PrIdTransfer             := TRUE,
           Start                    := TRUE,
           RetVal                   := #wRetVal);
Strt: NOP   0;
END_FUNCTION_BLOCK

FUNCTION_BLOCK FB 4119
TITLE =U111: Transfer Plant 11
AUTHOR : Woermann
FAMILY : BOTEC_F1
NAME : Sim
VERSION : 0.1


VAR_TEMP
  CIP : BOOL ;	//CIP active
  xTmp : BOOL ;	//Temporary BOOL (free for general use)
  iTmp : INT ;	//Temporary INT (free for general use)
  rTmp : REAL ;	//Temporary REAL (free for general use)
  UnitNo : INT ;	//Unit Number
END_VAR
BEGIN
NETWORK
TITLE =General

      SET   ;
// get unit number ----------------------------------------------------------
      L     DB4110.DBW    0;
      T     #UnitNo;

// CIP ----------------------------------------------------------------------
      L     DB4111.DBD   54;
      L     0;
      <D    ;
      =     #CIP;

NETWORK
TITLE =Actuator

      A     DB4111.DBX   17.3;
      =     DB5110.DBX 1465.3;
      =     DB5110.DBX 1545.3;
      =     DB5110.DBX 1945.3;
      =     DB5110.DBX 2025.3;
      =     DB5110.DBX 2105.3;
      =     DB5110.DBX 2185.3;
      =     DB5110.DBX 2265.3;
      =     DB5110.DBX 2345.3;
      =     DB5110.DBX 2425.3;
      =     DB5110.DBX 2505.3;
      =     DB5110.DBX 2585.3;
      =     DB5110.DBX 2665.3;
      =     DB5110.DBX 2745.3;
      =     DB5110.DBX 2825.3;
      =     DB5110.DBX 2905.3;
      =     DB5110.DBX 2985.3;


NETWORK
TITLE =Special Input

      A     DB4111.DBX   17.3;
      =     DB5111.DBX  561.3;

NETWORK
TITLE =Counter

      A     DB4111.DBX   17.3;
      A     M    101.0;


      CLR   ;
NETWORK
TITLE =Analog Input

      A     DB4111.DBX   17.3;

NETWORK
TITLE =Universal Value

      A     DB4111.DBX   17.3;
//      =     "U111UnVD".unv001.Sim;
//      =     "U111UnVD".unv002.Sim;
//      =     "U111UnVD".unv003.Sim;
//      =     "U111UnVD".unv004.Sim;

NETWORK
TITLE =PID

      A     DB4111.DBX   17.3;

NETWORK
TITLE =Message

      A     DB4111.DBX   17.3;
//      =     "U111MsgD".msg001.Sim;
//      =     "U111MsgD".msg002.Sim;
//      =     "U111MsgD".msg003.Sim;

NETWORK
TITLE =VLT

      A     DB4111.DBX   17.3;

END_FUNCTION_BLOCK

FUNCTION_BLOCK FB 4125
TITLE =U112: Transfer Plant 12
FAMILY : BOTEC_F1
NAME : Comm
VERSION : 0.1


VAR_TEMP
  iRetVal : INT ;	//return value as integer
  wRetVal : WORD ;	//return value as word
  Run : BOOL ;	//Unit in "RUN" mode
  EStopOK : BOOL ;	//Emergency Stop OK
  CIP : BOOL ;	//CIP Program Selected
  ComCIP : BOOL ;	//Communication with CIP Active
  xTmp : BOOL ;	//Temporary BOOL (free for general use)
  iTmp : INT ;	//Temporary INT (free for general use)
  rTmp : REAL ;	//Temporary REAL (free for general use)
  dTmp : DINT ;	//Temporary DINT (free for general use)
  UnitNo : INT ;	//Unit Number
  EquipmentID : INT ;	//Equipment ID
  Prid : DINT ;	//Process ID
  SFM36 : STRUCT 	// CIP Pump Mode
   I00 : BOOL ;	// Off
   I01 : BOOL ;	// Flow
   I02 : BOOL ;	// Pressure
   I03 : BOOL ;	// Fix Speed
   I04 : BOOL ;
   I05 : BOOL ;
   I06 : BOOL ;
   I07 : BOOL ;
   I08 : BOOL ;
   I09 : BOOL ;
   I10 : BOOL ;
   I11 : BOOL ;
   I12 : BOOL ;
   I13 : BOOL ;
   I14 : BOOL ;
   I15 : BOOL ;
   I16 : BOOL ;
   I17 : BOOL ;
   I18 : BOOL ;
   I19 : BOOL ;
   I20 : BOOL ;
   I21 : BOOL ;
   I22 : BOOL ;
   I23 : BOOL ;
   I24 : BOOL ;
   I25 : BOOL ;
   I26 : BOOL ;
   I27 : BOOL ;
   I28 : BOOL ;
   I29 : BOOL ;
   I30 : BOOL ;
   I31 : BOOL ;
  END_STRUCT ;
END_VAR
BEGIN
NETWORK
TITLE =general

      SET   ;

// unit & equipment number ---------------------------------------------------
      L     DB4120.DBW    0;
      T     #UnitNo;

      L     DB4125.DBW   14;
      L     1000;
      *I    ;
      L     #UnitNo;
      +I    ;
      T     #EquipmentID;

// CIP ----------------------------------------------------------------------
      L     DB4125.DBW   18;
      L     0;
      <I    ;
      =     #CIP;

// Communicating Units-------------------------------------------------------
      L     DB4125.DBD   10;
      L     DB4125.DBD  106;
      ==D   ;
      =     #ComCIP;

// emergency OK -------------------------------------------------------------
      A     DB4125.DBX   75.0; //General Emergency Stop OK
      =     #EStopOK;

NETWORK
TITLE =remote start

      SET   ;
      A     DB4121.DBX   66.2;
      A     DB4121.DBX   15.0;
      A     DB4121.DBX   17.4;
      JCN   Strt;
      L     DB4125.DBD   10;
      L     L#-1; // Prid negative to start on its own
      T     #Prid;

      CALL FC    48 (
           UnitNo                   := #UnitNo,
           PrId                     := #Prid,
           Run                      := DB4121.DBX   17.4,
           PrIdTransfer             := TRUE,
           Start                    := TRUE,
           RetVal                   := #wRetVal);
Strt: NOP   0;

// Start von Sirupraum (VP3)
      AN    DB1995.DBX 1368.7;
      A     DB1995.DBX 1368.0;
      A     DB4121.DBX   15.0;
      A     DB4121.DBX   17.4;
      JCN   Str2;
      L     DB1995.DBD 1354;
      T     #Prid;

      CALL FC    48 (
           UnitNo                   := #UnitNo,
           PrId                     := #Prid,
           Run                      := DB4121.DBX   17.4,
           PrIdTransfer             := TRUE,
           Start                    := TRUE,
           RetVal                   := #wRetVal);
Str2: NOP   0;

NETWORK
TITLE =
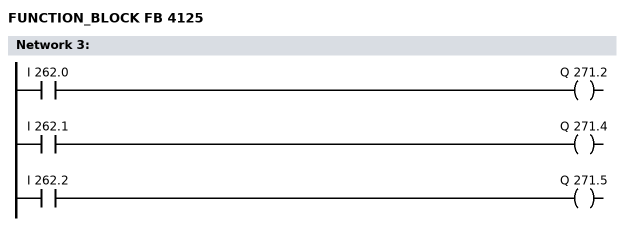



// Signale Panel an Mixer
      A     I    262.0;
      =     Q    271.2;
      A     I    262.1;
      =     Q    271.4;
      A     I    262.2;
      =     Q    271.5;


END_FUNCTION_BLOCK

FUNCTION_BLOCK FB 4129
TITLE =U112: Transfer Plant 12
AUTHOR : Woermann
FAMILY : BOTEC_F1
NAME : Sim
VERSION : 0.1


VAR_TEMP
  CIP : BOOL ;	//CIP active
  xTmp : BOOL ;	//Temporary BOOL (free for general use)
  iTmp : INT ;	//Temporary INT (free for general use)
  rTmp : REAL ;	//Temporary REAL (free for general use)
  UnitNo : INT ;	//Unit Number
END_VAR
BEGIN
NETWORK
TITLE =General

      SET   ;
// get unit number ----------------------------------------------------------
      L     DB4120.DBW    0;
      T     #UnitNo;

// CIP ----------------------------------------------------------------------
      L     DB4121.DBD   54;
      L     0;
      <D    ;
      =     #CIP;

NETWORK
TITLE =Actuator

      A     DB4121.DBX   17.3;
      =     DB5120.DBX  425.3;
      =     DB5120.DBX  505.3;
      =     DB5120.DBX  585.3;
      =     DB5120.DBX  665.3;
      =     DB5120.DBX  745.3;
      =     DB5120.DBX  825.3;
      =     DB5120.DBX  905.3;
      =     DB5120.DBX  985.3;
      =     DB5120.DBX 1065.3;
      =     DB5120.DBX 1145.3;
      =     DB5120.DBX 1225.3;
      =     DB5120.DBX 1305.3;
      =     DB5120.DBX 1385.3;
      =     DB5120.DBX 1465.3;
//      =     "U112ActD".A12_MOLCH_A12_L.Sim;
      =     DB5120.DBX 3145.3;
      =     DB5120.DBX 3225.3;
      =     DB5120.DBX 3305.3;

NETWORK
TITLE =Special Input

      A     DB4121.DBX   17.3;
      =     DB5121.DBX  441.3;
      =     DB5121.DBX  681.3;
      =     DB5121.DBX  741.3;
      =     DB5121.DBX 1041.3;
      =     DB5121.DBX 1101.3;
      =     DB5121.DBX 1161.3;
      =     DB5121.DBX 1221.3;
      =     DB5121.DBX 1281.3;
      =     DB5121.DBX 1341.3;
      =     DB5121.DBX 1461.3;
      =     DB5121.DBX 1521.3;
      =     DB5121.DBX 1581.3;
      =     DB5121.DBX 1641.3;
      =     DB5121.DBX 1701.3;
      =     DB5121.DBX 1761.3;
      =     DB5121.DBX 1821.3;
      =     DB5121.DBX 1881.3;
      =     DB5121.DBX 1941.3;


NETWORK
TITLE =Counter

      A     DB4121.DBX   17.3;
      A     M    101.0;


      CLR   ;
NETWORK
TITLE =Analog Input

      A     DB4121.DBX   17.3;

NETWORK
TITLE =Universal Value

      A     DB4121.DBX   17.3;
//      =     "U112UnVD".unv001.Sim;
//      =     "U112UnVD".unv002.Sim;
//      =     "U112UnVD".unv003.Sim;
//      =     "U112UnVD".unv004.Sim;

NETWORK
TITLE =PID

      A     DB4121.DBX   17.3;

NETWORK
TITLE =Message

      A     DB4121.DBX   17.3;
//      =     "U112MsgD".msg001.Sim;
//      =     "U112MsgD".msg002.Sim;
//      =     "U112MsgD".msg003.Sim;

NETWORK
TITLE =VLT

      A     DB4121.DBX   17.3;

END_FUNCTION_BLOCK

FUNCTION_BLOCK FB 4145
TITLE =U114: Transfer Plant 14
FAMILY : BOTEC_F1
NAME : Comm
VERSION : 0.1


VAR_TEMP
  iRetVal : INT ;	//return value as integer
  wRetVal : WORD ;	//return value as word
  Run : BOOL ;	//Unit in "RUN" mode
  EStopOK : BOOL ;	//Emergency Stop OK
  CIP : BOOL ;	//CIP Program Selected
  ComCIP : BOOL ;	//Communication with CIP Active
  xTmp : BOOL ;	//Temporary BOOL (free for general use)
  iTmp : INT ;	//Temporary INT (free for general use)
  rTmp : REAL ;	//Temporary REAL (free for general use)
  dTmp : DINT ;	//Temporary DINT (free for general use)
  UnitNo : INT ;	//Unit Number
  EquipmentID : INT ;	//Equipment ID
  Prid : DINT ;	//Process ID
  SFM36 : STRUCT 	// CIP Pump Mode
   I00 : BOOL ;	// Off
   I01 : BOOL ;	// Flow
   I02 : BOOL ;	// Pressure
   I03 : BOOL ;	// Fix Speed
   I04 : BOOL ;
   I05 : BOOL ;
   I06 : BOOL ;
   I07 : BOOL ;
   I08 : BOOL ;
   I09 : BOOL ;
   I10 : BOOL ;
   I11 : BOOL ;
   I12 : BOOL ;
   I13 : BOOL ;
   I14 : BOOL ;
   I15 : BOOL ;
   I16 : BOOL ;
   I17 : BOOL ;
   I18 : BOOL ;
   I19 : BOOL ;
   I20 : BOOL ;
   I21 : BOOL ;
   I22 : BOOL ;
   I23 : BOOL ;
   I24 : BOOL ;
   I25 : BOOL ;
   I26 : BOOL ;
   I27 : BOOL ;
   I28 : BOOL ;
   I29 : BOOL ;
   I30 : BOOL ;
   I31 : BOOL ;
  END_STRUCT ;
END_VAR
BEGIN
NETWORK
TITLE =general

      SET   ;

// unit & equipment number ---------------------------------------------------
      L     DB4140.DBW    0;
      T     #UnitNo;

      L     DB4145.DBW   14;
      L     1000;
      *I    ;
      L     #UnitNo;
      +I    ;
      T     #EquipmentID;

// CIP ----------------------------------------------------------------------
      L     DB4145.DBW   18;
      L     0;
      <I    ;
      =     #CIP;

// Communicating Units-------------------------------------------------------
      L     DB4145.DBD   10;
      L     DB4145.DBD  106;
      ==D   ;
      =     #ComCIP;

// emergency OK -------------------------------------------------------------
      A     DB4145.DBX   75.0; //General Emergency Stop OK
      =     #EStopOK;

NETWORK
TITLE =remote start
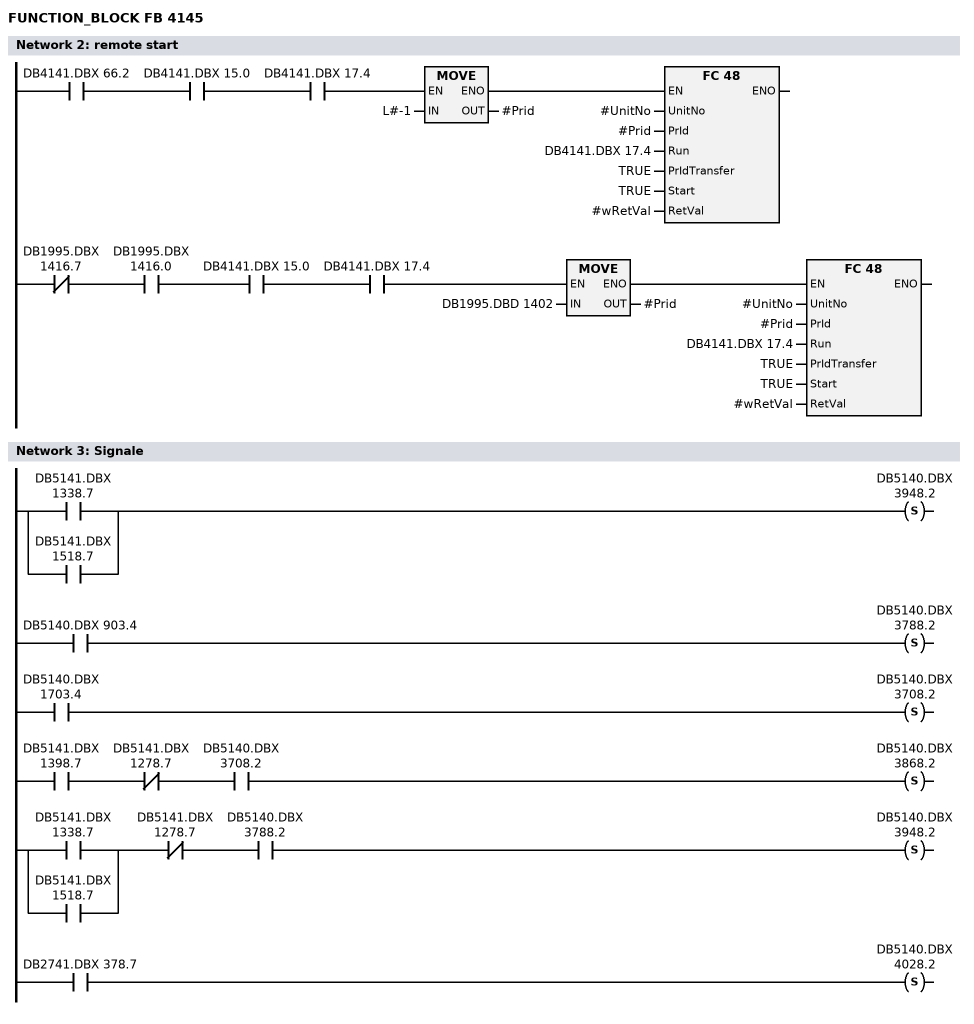

      SET   ;
      A     DB4141.DBX   66.2;
      A     DB4141.DBX   15.0;
      A     DB4141.DBX   17.4;
      JCN   Strt;
      L     L#-1; // Prid negative to start on its own
      T     #Prid;

      CALL FC    48 (
           UnitNo                   := #UnitNo,
           PrId                     := #Prid,
           Run                      := DB4141.DBX   17.4,
           PrIdTransfer             := TRUE,
           Start                    := TRUE,
           RetVal                   := #wRetVal);
Strt: NOP   0;

// Start von Sirupraum (VP3)
      AN    DB1995.DBX 1416.7;
      A     DB1995.DBX 1416.0;
      A     DB4141.DBX   15.0;
      A     DB4141.DBX   17.4;
      JCN   Str2;
      L     DB1995.DBD 1402;
      T     #Prid;

      CALL FC    48 (
           UnitNo                   := #UnitNo,
           PrId                     := #Prid,
           Run                      := DB4141.DBX   17.4,
           PrIdTransfer             := TRUE,
           Start                    := TRUE,
           RetVal                   := #wRetVal);
Str2: NOP   0;

NETWORK
TITLE =Signale


// Schwenkbogen auf CIP
      A     DB5141.DBX 1338.7;
      O     DB5141.DBX 1518.7;
      S     DB5140.DBX 3948.2;

// Molch im Sirupraum
      A     DB5140.DBX  903.4;
      S     DB5140.DBX 3788.2;

// Molch an der Anlage
      A     DB5140.DBX 1703.4;
      S     DB5140.DBX 3708.2;

// Bereit für Produktion
      A     DB5141.DBX 1398.7;
      AN    DB5141.DBX 1278.7;
      A     DB5140.DBX 3708.2;
      S     DB5140.DBX 3868.2;

// Bereit für CIP
      A     DB5141.DBX 1338.7;
      O     DB5141.DBX 1518.7;
      AN    DB5141.DBX 1278.7;
      A     DB5140.DBX 3788.2;
      S     DB5140.DBX 3948.2;

// Sirupanforderung
      A     DB2741.DBX  378.7;
      S     DB5140.DBX 4028.2;




END_FUNCTION_BLOCK

FUNCTION_BLOCK FB 4149
TITLE =U114: Transfer Plant 14
AUTHOR : Woermann
FAMILY : BOTEC_F1
NAME : Sim
VERSION : 0.1


VAR_TEMP
  CIP : BOOL ;	//CIP active
  xTmp : BOOL ;	//Temporary BOOL (free for general use)
  iTmp : INT ;	//Temporary INT (free for general use)
  rTmp : REAL ;	//Temporary REAL (free for general use)
  UnitNo : INT ;	//Unit Number
END_VAR
BEGIN
NETWORK
TITLE =General

      SET   ;
// get unit number ----------------------------------------------------------
      L     DB4140.DBW    0;
      T     #UnitNo;

// CIP ----------------------------------------------------------------------
      L     DB4141.DBD   54;
      L     0;
      <D    ;
      =     #CIP;

NETWORK
TITLE =Actuator

      A     DB4141.DBX   17.3;
      =     DB5140.DBX  425.3;
      =     DB5140.DBX  505.3;
      =     DB5140.DBX  585.3;
      =     DB5140.DBX  665.3;
      =     DB5140.DBX  745.3;
      =     DB5140.DBX  825.3;
      =     DB5140.DBX  905.3;
      =     DB5140.DBX  985.3;
      =     DB5140.DBX 1065.3;
      =     DB5140.DBX 1145.3;
      =     DB5140.DBX 1225.3;
      =     DB5140.DBX 1305.3;
      =     DB5140.DBX 2665.3;
      =     DB5140.DBX 2745.3;
      =     DB5140.DBX 2825.3;
      =     DB5140.DBX 2905.3;
      =     DB5140.DBX 3065.3;
      =     DB5140.DBX 3145.3;
      =     DB5140.DBX 3225.3;
      =     DB5140.DBX 3305.3;

NETWORK
TITLE =Special Input

      A     DB4141.DBX   17.3;
      =     DB5141.DBX  681.3;
      =     DB5141.DBX  741.3;
      =     DB5141.DBX 1041.3;
      =     DB5141.DBX 1221.3;
      =     DB5141.DBX 1281.3;
      =     DB5141.DBX 1341.3;
      =     DB5141.DBX 1461.3;
      =     DB5141.DBX 1521.3;
      =     DB5141.DBX 1581.3;
      =     DB5141.DBX 1641.3;
      =     DB5141.DBX 1701.3;
      =     DB5141.DBX 1761.3;
      =     DB5141.DBX 1821.3;
      =     DB5141.DBX 1881.3;
      =     DB5141.DBX 1941.3;


NETWORK
TITLE =Counter

      A     DB4141.DBX   17.3;
      A     M    101.0;


      CLR   ;
NETWORK
TITLE =Analog Input

      A     DB4141.DBX   17.3;

NETWORK
TITLE =Universal Value

      A     DB4141.DBX   17.3;
//      =     "U114UnVD".unv001.Sim;
//      =     "U114UnVD".unv002.Sim;
//      =     "U114UnVD".unv003.Sim;
//      =     "U114UnVD".unv004.Sim;

NETWORK
TITLE =PID

      A     DB4141.DBX   17.3;

NETWORK
TITLE =Message

      A     DB4141.DBX   17.3;
//      =     "U114MsgD".msg001.Sim;
//      =     "U114MsgD".msg002.Sim;
//      =     "U114MsgD".msg003.Sim;

NETWORK
TITLE =VLT

      A     DB4141.DBX   17.3;

END_FUNCTION_BLOCK

FUNCTION_BLOCK FB 4215
TITLE =U121: Planung Transfer VE1
FAMILY : BOTEC_F1
NAME : U121Comm
VERSION : 0.1


